(* CoDeSys 2.3 project: cy-wg-03_030.pro *)
(* Title: cy-003-wg (SanFelice) *)
(* Author: Andrea Ravasio *)
(* Libraries: serial_interface_01.lib 22.4.13 12:50:14, SerComm.lib 31.5.11 08:54:36, MBus_03.lib 22.7.15 16:25:47, Util.lib 26.9.14 10:12:46, Visual.lib 2.12.10 14:48:34, WagoLibIdent.lib 25.2.13 11:12:16, WagoLibStatus.lib 2.12.10 14:48:32, SysLibFile.lib 2.12.10 14:48:34, SysLibRtc.lib 2.12.10 14:48:32, SysLibSockets.lib 10.2.11 09:20:54, SysLibEvent.lib 2.12.10 14:48:34, SysLibPlcCtrl.lib 2.12.10 14:48:32, Standard.lib 2.12.10 14:48:34, SYSLIBCALLBACK.LIB 2.12.10 14:48:32 *)

(* PLC configuration (modules and I/O channels)
K-Bus [K_Bus] node 0, in %IB0 out %QB0
  0750-0402 4 DI 24 V DC 3.0ms [Type_1_4_Channels] node 0, in %IB24 out %QB4 {INTTypePAAssignment = PLC; INTTypeModule = plugged}
    VPN_ST2 AT %IX12.0 [BOOLOnX_I] Ch_1 Digital input
    KEY_QE_ST AT %IX12.1 [BOOLOnX_I] Ch_2 Digital input
    SCA01_5_DI AT %IX12.2 [BOOLOnX_I] Ch_3 Digital input
    PORT01_DI AT %IX12.3 [BOOLOnX_I] Ch_4 Digital input
  0750-0402 4 DI 24 V DC 3.0ms [Type_1_4_Channels] node 1, in %IB24 out %QB4 {INTTypePAAssignment = PLC; INTTypeModule = plugged}
    GAS02_DI AT %IX12.4 [BOOLOnX_I] Ch_1 Digital input
    GAS01_DI AT %IX12.5 [BOOLOnX_I] Ch_2 Digital input
    SCA01_6_DI AT %IX12.6 [BOOLOnX_I] Ch_3 Digital input
    SCA02_1_DI AT %IX12.7 [BOOLOnX_I] Ch_4 Digital input
  0750-1506 8DI / 8DO 24V DC 0.5A [Type_34_8_Channels] node 2, in %IX12.4 out %QB4 {INTTypePAAssignment = PLC; INTTypeModule = plugged}
    SCA02_2_DI AT %IX12.8 [BOOLOnX_I] Ch_1 Digital input
    SCA01_1_DO AT %QX2.0 [BOOLOnX_Q] Ch_1 Digital output
    SCA02_3_DI AT %IX12.9 [BOOLOnX_I] Ch_2 Digital input
    SCA01_2_DO AT %QX2.1 [BOOLOnX_Q] Ch_2 Digital output
    SCA02_4_DI AT %IX12.10 [BOOLOnX_I] Ch_3 Digital input
    SCA01_3_DO AT %QX2.2 [BOOLOnX_Q] Ch_3 Digital output
    SCA02_5_DI AT %IX12.11 [BOOLOnX_I] Ch_4 Digital input
    SCA01_4_DO AT %QX2.3 [BOOLOnX_Q] Ch_4 Digital output
    SCA02_6_DI AT %IX12.12 [BOOLOnX_I] Ch_5 Digital input
    AT %QX2.4 [BOOLOnX_Q] Ch_5 Digital output
    SCA02_7_DI AT %IX12.13 [BOOLOnX_I] Ch_6 Digital input
    AT %QX2.5 [BOOLOnX_Q] Ch_6 Digital output
    SCA02_8_DI AT %IX12.14 [BOOLOnX_I] Ch_7 Digital input
    AT %QX2.6 [BOOLOnX_Q] Ch_7 Digital output
    SCA02_9_DI AT %IX12.15 [BOOLOnX_I] Ch_8 Digital input
    AT %QX2.7 [BOOLOnX_Q] Ch_8 Digital output
  0750-1506 8DI / 8DO 24V DC 0.5A [Type_34_8_Channels] node 3, in %IB25 out %QB4 {INTTypePAAssignment = PLC; INTTypeModule = plugged}
    SCA03_1_DI AT %IX13.0 [BOOLOnX_I] Ch_1 Digital input
    AT %QX2.8 [BOOLOnX_Q] Ch_1 Digital output
    SCA03_2_DI AT %IX13.1 [BOOLOnX_I] Ch_2 Digital input
    AT %QX2.9 [BOOLOnX_Q] Ch_2 Digital output
    SCA03_3_DI AT %IX13.2 [BOOLOnX_I] Ch_3 Digital input
    AT %QX2.10 [BOOLOnX_Q] Ch_3 Digital output
    SCA03_4_DI AT %IX13.3 [BOOLOnX_I] Ch_4 Digital input
    AT %QX2.11 [BOOLOnX_Q] Ch_4 Digital output
    SCA03_5_DI AT %IX13.4 [BOOLOnX_I] Ch_5 Digital input
    AT %QX2.12 [BOOLOnX_Q] Ch_5 Digital output
    SCA03_6_DI AT %IX13.5 [BOOLOnX_I] Ch_6 Digital input
    AT %QX2.13 [BOOLOnX_Q] Ch_6 Digital output
    SCA03_7_DI AT %IX13.6 [BOOLOnX_I] Ch_7 Digital input
    AT %QX2.14 [BOOLOnX_Q] Ch_7 Digital output
    SCA03_8_DI AT %IX13.7 [BOOLOnX_I] Ch_8 Digital input
    AT %QX2.15 [BOOLOnX_Q] Ch_8 Digital output
  0750-1506 8DI / 8DO 24V DC 0.5A [Type_34_8_Channels] node 4, in %IB26 out %QB5 {INTTypePAAssignment = PLC; INTTypeModule = plugged}
    SCA03_9_DI AT %IX13.8 [BOOLOnX_I] Ch_1 Digital input
    AT %QX3.0 [BOOLOnX_Q] Ch_1 Digital output
    SCA03_10_DI AT %IX13.9 [BOOLOnX_I] Ch_2 Digital input
    AT %QX3.1 [BOOLOnX_Q] Ch_2 Digital output
    SCA03_11_DI AT %IX13.10 [BOOLOnX_I] Ch_3 Digital input
    AT %QX3.2 [BOOLOnX_Q] Ch_3 Digital output
    SCA03_12_DI AT %IX13.11 [BOOLOnX_I] Ch_4 Digital input
    AT %QX3.3 [BOOLOnX_Q] Ch_4 Digital output
    SCA03_13_DI AT %IX13.12 [BOOLOnX_I] Ch_5 Digital input
    AT %QX3.4 [BOOLOnX_Q] Ch_5 Digital output
    SCA03_14_DI AT %IX13.13 [BOOLOnX_I] Ch_6 Digital input
    AT %QX3.5 [BOOLOnX_Q] Ch_6 Digital output
    SCA03_15_DI AT %IX13.14 [BOOLOnX_I] Ch_7 Digital input
    AT %QX3.6 [BOOLOnX_Q] Ch_7 Digital output
    SCA03_16_DI AT %IX13.15 [BOOLOnX_I] Ch_8 Digital input
    AT %QX3.7 [BOOLOnX_Q] Ch_8 Digital output
  0750-1506 8DI / 8DO 24V DC 0.5A [Type_34_8_Channels] node 5, in %IB27 out %QB6 {INTTypePAAssignment = PLC; INTTypeModule = plugged}
    SCA03_17_DI AT %IX14.0 [BOOLOnX_I] Ch_1 Digital input
    AT %QX3.8 [BOOLOnX_Q] Ch_1 Digital output
    SCA03_18_DI AT %IX14.1 [BOOLOnX_I] Ch_2 Digital input
    AT %QX3.9 [BOOLOnX_Q] Ch_2 Digital output
    SCA03_19_DI AT %IX14.2 [BOOLOnX_I] Ch_3 Digital input
    AT %QX3.10 [BOOLOnX_Q] Ch_3 Digital output
    SCA03_20_DI AT %IX14.3 [BOOLOnX_I] Ch_4 Digital input
    AT %QX3.11 [BOOLOnX_Q] Ch_4 Digital output
    SCA03_21_DI AT %IX14.4 [BOOLOnX_I] Ch_5 Digital input
    AT %QX3.12 [BOOLOnX_Q] Ch_5 Digital output
    SCA03_22_DI AT %IX14.5 [BOOLOnX_I] Ch_6 Digital input
    AT %QX3.13 [BOOLOnX_Q] Ch_6 Digital output
    AT %IX14.6 [BOOLOnX_I] Ch_7 Digital input
    TEST1 AT %QX3.14 [BOOLOnX_Q] Ch_7 Digital output
    AT %IX14.7 [BOOLOnX_I] Ch_8 Digital input
    TEST2 AT %QX3.15 [BOOLOnX_Q] Ch_8 Digital output
  0750-0464#02 2/4 AI RTD / ADJ./ HA [Type_44_2_Channels] node 6, in %IB20 out %QB0 {INTTypePAAssignment = PLC; INTTypeModule = plugged}
    TT_S01 AT %IW0 [INTOnW_I] Ch_1 signed Input value
    AT %IW1 [INTOnW_I] Ch_2 signed Input value
  0750-0472 2 AI 0-20mA 16 Bit S.E. [Type_8_2_Channels] node 7, in %IB20 out %QB0 {INTTypePAAssignment = PLC; INTTypeModule = plugged}
    TT_S07 AT %IW2 [WORDOnW_I] I 1: Analog Input
    TT_S06 AT %IW3 [WORDOnW_I] I 2: Analog Input
  0750-0472 2 AI 0-20mA 16 Bit S.E. [Type_8_2_Channels] node 8, in %IB24 out %QB0 {INTTypePAAssignment = PLC; INTTypeModule = plugged}
    TT_S05 AT %IW4 [WORDOnW_I] I 1: Analog Input
    TT_S04 AT %IW5 [WORDOnW_I] I 2: Analog Input
  0750-0472 2 AI 0-20mA 16 Bit S.E. [Type_8_2_Channels] node 9, in %IB28 out %QB0 {INTTypePAAssignment = PLC; INTTypeModule = plugged}
    TT_S03 AT %IW6 [WORDOnW_I] I 1: Analog Input
    TT_S02 AT %IW7 [WORDOnW_I] I 2: Analog Input
  0750-0472 2 AI 0-20mA 16 Bit S.E. [Type_8_2_Channels] node 10, in %IB32 out %QB0 {INTTypePAAssignment = PLC; INTTypeModule = plugged}
    PORT01_AI AT %IW8 [WORDOnW_I] I 1: Analog Input
    AT %IW9 [WORDOnW_I] I 2: Analog Input
  0750-0650/0003-0000#03 RS 232 C Interface (Adjustable), 3 Byte [Type_21_1_Channels] node 0, in %IB36 out %QB0 {INTTypePAAssignment = PLC; INTTypeModule = plugged}
    AT %IX10.0 [BOOLOnX_I] Transmission acknowledgement
    AT %IX10.1 [BOOLOnX_I] Reception request
    AT %IX10.2 [BOOLOnX_I] Initialization acknowledgement
    AT %IX10.3 [BOOLOnX_I] Input buffer is full
    AT %IX10.4 [BOOLOnX_I] Number of received characters Bit 0
    AT %IX10.5 [BOOLOnX_I] Number of received characters Bit 1
    AT %IX10.6 [BOOLOnX_I] Number of received characters Bit 2
    AT %IB21 [BYTEOnB_I] Input data Byte 0
    AT %IB22 [BYTEOnB_I] Input data Byte 1
    AT %IB23 [BYTEOnB_I] Input data Byte 2
    AT %QX0.0 [BOOLOnX_Q] Transmission request
    AT %QX0.1 [BOOLOnX_Q] Reception acknowledgement
    AT %QX0.2 [BOOLOnX_Q] Initialization request
    AT %QX0.4 [BOOLOnX_Q] Number of characters Bit 0
    AT %QX0.5 [BOOLOnX_Q] Number of characters Bit 1
    AT %QX0.6 [BOOLOnX_Q] Number of characters Bit 2
    AT %QB1 [BYTEOnB_Q] Output data Byte 0
    AT %QB2 [BYTEOnB_Q] Output data Byte 1
    AT %QB3 [BYTEOnB_Q] Output data Byte 2
Fieldbus variables [FB_VARS] node 1, in %IB0 out %QB0
Flag variables [FLAG_VARS] node 2, in %IB0 out %QB0
Modbus-Master [MB_MASTER] node 3, in %IB0 out %QB0
*)

(* Task configuration *)
TASK FastCounter (PRIORITY := 5, INTERVAL := T#3ms);
	PLC_FAST_CTR();
END_TASK
TASK Main (PRIORITY := 10); (* freewheeling *)
	PLC_PRG();
END_TASK

(* Global variable list: Global_Constants *)
VAR_GLOBAL CONSTANT

	Plant_NAME			: STRING :='cySN:3 cyVER:30 - San Felice';
	Plant_SN			: DWORD :=3;   		(* S/N Impianto di telecontrollo *)
	Plant_SW_VER		: WORD  :=30;		(* Versione SW installata *)

	(* Parameters *)
	Plant_DefaultTAmb	: INT	:=-9999;	(* [.1°C] Temperatura ambiente di default in caso di rottura sonda *)

	(* Filesystem *)
	FilesPath  			: STRING :='S:\';

	(* TCP Logger *)
	Logger_SERVER		: STRING:='';
	Logger_IP			: STRING:='192.168.100.3';
	Logger_PORT			: WORD  :=80;
	Logger_GETSTART		: STRING:='GET /cygmsrv/hsgm.ashx?';
	Logger_GETEND		: STRING:='$R$N$R$N';
	Logger_CHECK		: STRING:='True';
	Logger_CRLF			: STRING:='$R$N';
	Logger_DataFile		: STRING:='S:\LOG.DAT';
	Logger_DataFileOld	: STRING:='S:\LOG.BCK';
	Logger_IndexFile	: STRING:='S:\LOG.IDX';
	Logger_ConnRetries	: BYTE:=5;
	Logger_RecoverMsgs	: BYTE:=100;

	(* TCP Remote *)
	Remote_PORT			: WORD  :=10;
	Remote_WELCOME		: STRING:='Connected$R$N';
	Remote_OK			: STRING:='OK$R$N';
	Remote_ERROR		: STRING:='ERROR$R$N';

	(* TCP Sockets *)
	MAX_SEND_TCP_SERVER					 : DWORD:=1500;(*60000*)
	MAX_RECEIVE_TCP_SERVER				 : DWORD:=3000;
	MAX_RECEIVE_TCP_SERVER_SOCKET	 	 : DWORD:=1500;
	MAX_SEND_TCP_CLIENT					 : DWORD:=3000;(*15000*)
	MAX_RECEIVE_TCP_CLIENT				 : DWORD:=1500;
	MAX_RECEIVE_TCP_CLIENT_SOCKET		 : DWORD:=1500;
	MAX_RECEIVE_UDP_SERVER				 : INT  :=1472;
	MAX_RECEIVE_UDP_CLIENT				 : INT  :=1472;
	CONNECT_WATCHDOG_TIME				 : TIME :=t#10s;

	(* VISU COLORS *)
	COLOR_RED 			: DWORD:=16#2020F0;
	COLOR_YELLOW		: DWORD:=16#20F0F0;
	COLOR_GREEN			: DWORD:=16#20F020;
	COLOR_GREEN_OFF 	: DWORD:=16#006000;
	COLOR_LBLUE			: DWORD:=16#F0F080;
	COLOR_GREY			: DWORD:=16#C0C0C0;

END_VAR

(* Global variable list: Global_Retain *)
VAR_GLOBAL RETAIN PERSISTENT

	PortataTotalePORT01		: DINT;
	ConteggioTotalePORT01	: DINT;
	PortataTotaleGAS01		: DINT;
	ConteggioTotaleGAS01	: DINT;
	PortataTotaleGAS02		: DINT;
	ConteggioTotaleGAS02	: DINT;

	CTB250_ENERGY_WH		: REAL;
	CTB250_ENERGY			: DWORD; (* 10^-2 MWh *)

	Mode_Manual : BOOL := FALSE;
END_VAR

(* Global variable list: Global_Variables *)
VAR_GLOBAL

	SYS    : typ_SYS;
	T_AMB  : INT;

	TPV01  : obj_TPV		:= ( ID:=1,
								 IN_EMIN:=-600 , IN_EMAX:=2500 ,
								 IN_WMIN:=-500 , IN_WMAX:=600 ); (* T_S01 *)

	TPV02  : obj_TPV_SENS	:= ( ID:=2 ,
											SogliaHL:=4096 ,   	 	(* Soglia Sonda Aperta = 2,5mA *)
											SogliaHH:=32767,	 	(* Soglia Sonda CC = 20mA *)
											SogliaWL:=10, 			(* Soglia WRN Bassa  = 10°C *)
											SogliaWH:=120,			(* Soglia WRN Alta  = 120°C *)
											PuntoMinX:=0, 		    (* Scalatura Minima vedi data di targa sonda 0°C *)
											PuntoMaxX:=160,			(* Scalatura Massima Vedi data di targa Sonda 160°C *)
											PuntoMinY:=6553,		(* Valore minimio per scalatura = 4mA *)
											PuntoMaxY:=32767,		(* Valore Massimo per Scalatura = 20mA *)
											Decimali:=1); 			(* Decimali da ottenere durante la scalatura *)
	TPV03  : obj_TPV_SENS	:= ( ID:=3 ,
											SogliaHL:=4096 ,   	 	(* Soglia Sonda Aperta = 2,5mA *)
											SogliaHH:=32767,	 	(* Soglia Sonda CC = 20mA *)
											SogliaWL:=10, 			(* Soglia WRN Bassa  = 10°C *)
											SogliaWH:=120,			(* Soglia WRN Alta  = 120°C *)
											PuntoMinX:=0, 		    (* Scalatura Minima vedi data di targa sonda 0°C *)
											PuntoMaxX:=160,			(* Scalatura Massima Vedi data di targa Sonda 160°C *)
											PuntoMinY:=6553,		(* Valore minimio per scalatura = 4mA *)
											PuntoMaxY:=32767,		(* Valore Massimo per Scalatura = 20mA *)
											Decimali:=1); 			(* Decimali da ottenere durante la scalatura *)

	TPV04  : obj_TPV_SENS	:= ( ID:=4 ,
											SogliaHL:=4096 ,   	 	(* Soglia Sonda Aperta = 2,5mA *)
											SogliaHH:=32767,	 	(* Soglia Sonda CC = 20mA *)
											SogliaWL:=10, 			(* Soglia WRN Bassa  = 10°C *)
											SogliaWH:=120,			(* Soglia WRN Alta  = 120°C *)
											PuntoMinX:=0, 		    (* Scalatura Minima vedi data di targa sonda 0°C *)
											PuntoMaxX:=160,			(* Scalatura Massima Vedi data di targa Sonda 160°C *)
											PuntoMinY:=6553,		(* Valore minimio per scalatura = 4mA *)
											PuntoMaxY:=32767,		(* Valore Massimo per Scalatura = 20mA *)
											Decimali:=1); 			(* Decimali da ottenere durante la scalatura *)

	TPV05  : obj_TPV_SENS	:= ( ID:=5 ,
											SogliaHL:=4096 ,   	 	(* Soglia Sonda Aperta = 2,5mA *)
											SogliaHH:=32767,	 	(* Soglia Sonda CC = 20mA *)
											SogliaWL:=10, 			(* Soglia WRN Bassa  = 10°C *)
											SogliaWH:=120,			(* Soglia WRN Alta  = 120°C *)
											PuntoMinX:=0, 		    (* Scalatura Minima vedi data di targa sonda 0°C *)
											PuntoMaxX:=160,			(* Scalatura Massima Vedi data di targa Sonda 160°C *)
											PuntoMinY:=6553,		(* Valore minimio per scalatura = 4mA *)
											PuntoMaxY:=32767,		(* Valore Massimo per Scalatura = 20mA *)
											Decimali:=1); 			(* Decimali da ottenere durante la scalatura *)

	TPV06  : obj_TPV_SENS	:= ( ID:=6 ,
											SogliaHL:=4096 ,   	 	(* Soglia Sonda Aperta = 2,5mA *)
											SogliaHH:=32767,	 	(* Soglia Sonda CC = 20mA *)
											SogliaWL:=10, 			(* Soglia WRN Bassa  = 10°C *)
											SogliaWH:=120,			(* Soglia WRN Alta  = 120°C *)
											PuntoMinX:=0, 		    (* Scalatura Minima vedi data di targa sonda 0°C *)
											PuntoMaxX:=160,			(* Scalatura Massima Vedi data di targa Sonda 160°C *)
											PuntoMinY:=6553,		(* Valore minimio per scalatura = 4mA *)
											PuntoMaxY:=32767,		(* Valore Massimo per Scalatura = 20mA *)
											Decimali:=1); 			(* Decimali da ottenere durante la scalatura *)

	TPV07  : obj_TPV_SENS	:= ( ID:=7 ,
											SogliaHL:=4096 ,   	 	(* Soglia Sonda Aperta = 2,5mA *)
											SogliaHH:=32767,	 	(* Soglia Sonda CC = 20mA *)
											SogliaWL:=10, 			(* Soglia WRN Bassa  = 10°C *)
											SogliaWH:=120,			(* Soglia WRN Alta  = 120°C *)
											PuntoMinX:=0, 		    (* Scalatura Minima vedi data di targa sonda 0°C *)
											PuntoMaxX:=160,			(* Scalatura Massima Vedi data di targa Sonda 160°C *)
											PuntoMinY:=6553,		(* Valore minimio per scalatura = 4mA *)
											PuntoMaxY:=32767,		(* Valore Massimo per Scalatura = 20mA *)
											Decimali:=1); 			(* Decimali da ottenere durante la scalatura *)
	(* Misuratore di Portata *)
	PORT01  : obj_PORT	:=  ( ID:=1 ,
											TempoTimeOut:=T#2m,		(* PULSE - Minuti di attesa prima di segnalare WRN di inattività sulla linea *)
											SogliaHL:=4096,   	 	(* FLOW - Soglia Sonda Aperta = 2,5mA *)
											SogliaHH:=32767,	 	(* FLOW - Soglia Sonda CC = 20mA *)
											SogliaWL:=100000, 		(* FLOW - [E-3 m3/h] Soglia WRN Bassa *)
											SogliaWH:=700000,		(* FLOW - [E-3 m3/h] Soglia WRN Alta *)
											PuntoMinX:=0, 		    (* FLOW - [E-3 m3/h] Scalatura minima vedi data di targa sonda *)
											PuntoMaxX:=800000,		(* FLOW - [E-3 m3/h] Scalatura massima Vedi data di targa sonda *)
											PuntoMinY:=6553,		(* FLOW - Valore minimio per scalatura = 4mA *)
											PuntoMaxY:=32767		(* FLOW - Valore massimo per Scalatura = 20mA *)
											);

	(*  Contatori *)
	GAS01  : obj_GAS:=  (ID:=1,	Peso:=1 ,				(* Peso del'impulso *)
								TempoTimeOut:=T#15m		(* Minuti di attesa prima di segnalare WRN di inattività sulla linea *)
													  );
	GAS02  : obj_GAS:=  (ID:=2,	Peso:=1 ,				(* Peso del'impulso *)
								TempoTimeOut:=T#15m		(* Minuti di attesa prima di segnalare WRN di inattività sulla linea *)
													  );

	(* MBUS Contabilizers *)
	MBUS01 	  : obj_MBUS				:= ( ID:=1 , COM:=2 , BAUDRATE:=BAUD_2400 );
	CTBSCAN01 : obj_MBUS_CTB_SCANNER	:= ( ID:=1 );
	(*---- MBUS DEBUG ----*)
(*	COMx					: SERIAL_INTERFACE := (bCOM_PORT_NR		:= 2,
			cbBAUDRATE			:= BAUD_2400,
			cbsBYTESIZE			:= BS_8,
			cpPARITY			:= PARITY_EVEN,
			csSTOPBITS			:= STOPBITS_1,
			cfFLOW_CONTROL		:= NO_FLOW_CONTROL);
	RXBuf					: typRING_BUFFER;
	TXBuf					: ARRAY [0..16] OF BYTE;
	xINI					: BOOL;
	xSND					: BOOL;
	maddress : BYTE;
	mchk : BYTE;
	mt1 : BOOL;
	mt2 : BOOL;
	mt3 : BOOL;
*)

	(* Virtual contabilizers *)
	CTB250	  : obj_SW_CTB				:= ( ID:=250 );

	Logger : typ_Logger;

	(**** SIMULATION ONLY ****)
	(*...*)
END_VAR

(* Data type in Errors *)
TYPE en_Logger_ErrLev :
(
	EL_Log			:=0,
	EL_Wrn			:=1,
	EL_Alarm		:=2,
	EL_AlarmStop	:=3
);
END_TYPE

(* Data type in Errors *)
TYPE en_Logger_Status :
(
	S_Logger_UNKNOWN := 0,
	S_Logger_IDLE,
	S_Logger_WAITCONN,
	S_Logger_WAITTX,
	S_Logger_WAITRESP,
	S_Logger_ERROR
);
END_TYPE

(* Data type *)
TYPE en_SYS_Objects :
(
	EO_SYS		:=0,  (* PLC *)
	EO_VPN		:=1,  (* VPN *)
	EO_DOOR		:=2,  (* Door & access control *)

	EO_CAL		:=10, (* Caldaia *)
	EO_CIR		:=11, (* Circolatore *)
	EO_CRON		:=12, (* Crono-termostato *)
	EO_VRD		:=13, (* Valvola miscelatore pannelli *)
	EO_CTL		:=14, (* Contalitri *)
	EO_CTB		:=15, (* Contabilizzatore *)
	EO_TPV		:=16, (* Temperature probes values *)
	EO_PPV		:=17, (* Pressure probes values *)
	EO_PBV		:=18, (* Over-Pressure Alarms *)
	EO_TBV		:=19, (* Over-Temperature Alarms *)
	EO_PMV		:=20, (* Under-Pressure Alarms *)
	EO_GRU		:=21, (* Gruppo termico *)
	EO_PDC		:=22, (* Pompa di calore *)
	EO_SOL		:=23, (* Pannello solare termico *)
	EO_ESOL		:=24, (* Pannello solare fotovoltaico *)
	EO_GAS		:=25, (* Contatore GAS *)
	EO_PORT		:=26, (* Misuratore di portata *)
	EO_FPV		:=27, (* Flow probes values *)
	EO_ANZ		:=28,
	EO_SCA		:=29,

	EO_LON		:=1000, (* Bus - LON *)
	EO_MODBUS	:=1001, (* Bus - MODBUS *)
	EO_MBUS		:=1002  (* Bus - M-BUS *)
);
END_TYPE

(* Data type *)
TYPE en_SYS_Status :
(
	S_UNKNOWN  := 0,
	S_STARTUP,
	S_INIT_RTC,
	S_INIT_VAR,
	S_AUTOTEST,
	S_RUNNING,
	S_SHUTDOWN,
	S_HALT
);
END_TYPE

(* Data type in Errors *)
TYPE typ_Logger :
STRUCT
	Status		: en_Logger_Status;

	SendReq		: BOOL;
	SendIdx		: DWORD;
	SendData	: ARRAY [0..MAX_SEND_TCP_CLIENT] OF BYTE;
	SendLen		: DINT;

	TData		: ARRAY [0..MAX_SEND_TCP_CLIENT] OF BYTE;
	TLen		: DINT;

	LastIdxPos	: DWORD;

	(* Temporary variables used by objects *)
	s1			: STRING(256);
	i1			: WORD;

END_STRUCT
END_TYPE

(* Data type in Plant_Objects *)
TYPE typ_MBUS_CTBS :
STRUCT
	Present			: BOOL;
	Address			: DWORD;
	NodeError		: BYTE;

	Info			: typMBusInfo;
	Data_FTemp	 	: REAL; (* C *)
	Data_RTemp	 	: REAL; (* C *)
	Data_Flow	 	: REAL; (* m3ph *)
	Data_Power	 	: REAL; (* W *)
	Data_Energy 	: REAL; (* kWh *)

	Status_Log		: BYTE;
	Status_Vis		: DWORD;

END_STRUCT
END_TYPE

(* Data type *)
TYPE typ_SYS :
STRUCT
	Status			: en_SYS_Status;
	Warning			: BOOL;
	Alarm			: BOOL;
	AlarmStop		: BOOL;

	Time_LogString	: STRING;
	Time_Year		: WORD;
	Time_Month		: BYTE;
	Time_Day		: BYTE;

	Time_CT_DT		: DT;
	Time_CT_Day		: WORD;
	Time_CT_Quarter	: BYTE;

	LastLogs_Idx	: BYTE;
	LastLogs_Dat	: ARRAY[0..5] OF STRING;
	LastLogs_Msg	: ARRAY[0..5] OF STRING;

END_STRUCT
END_TYPE

(* Data type in Plant_Objects *)
TYPE typ_VisuStrutturaMbus :
STRUCT

	sdNodoPresente: STRING(16);
	sdEnergia: STRING(16);
	sdPotenza: STRING(16);
	sdVolume: STRING(16);
	sdFlow: STRING(16);
	sdTempIngresso: STRING(8);
	sdTempaUscita: STRING(8);
	sdTempDelta: STRING(8);

END_STRUCT
END_TYPE

(* POU PLC_FAST_CTR, ST *)
PROGRAM PLC_FAST_CTR
VAR
END_VAR
GAS01.Count(Contatore:=ConteggioTotaleGAS01, Totalizzatore:=PortataTotaleGAS01);
GAS02.Count(Contatore:=ConteggioTotaleGAS02, Totalizzatore:=PortataTotaleGAS02);
END_PROGRAM

(* POU PLC_PRG, ST *)
PROGRAM PLC_PRG
VAR
	Timer1: TON; (* Fast controls tick *)
	Timer2: TON; (* Plant control tick *)
	Timer3: TON; (* Logger timer *)

	t_sum : INT; (* Vars for dynamic means of working probes *)
	t_cnt : INT;
END_VAR
(******************************************************************************
 ****                           MAIN TASK CODE                             ****
 ******************************************************************************

	Network setup:
		IP  = 192.168.100.2 | MSK = 255.255.255.0 | GW = 192.168.100.1
		DNS = 192.168.100.1 | NTP = 193.168.100.3

	Editor setup:
		Project --> Options --> Editor --> Fonts --> Courier NEW / BOLD / 12

*)

(*==============================*)
(*===== Main status machine ====*)
(*==============================*)
Main_Stm();

(*=====================================*)
(*== Running common cycle operations ==*)
(*=====================================*)
IF SYS.Status>S_INIT_VAR THEN

	(* Execute M-BUS processes *)
	MBUS01();
	CTBSCAN01( MBUS:=MBUS01 );

	GAS01 ( GAS_DI:=GAS01_DI, Totalizzatore:=PortataTotaleGAS01, Contatore:=ConteggioTotaleGAS01 );
	GAS02 ( GAS_DI:=GAS02_DI, Totalizzatore:=PortataTotaleGAS02, Contatore:=ConteggioTotaleGAS02 );

(*	COMx(	ptSEND_BUFFER		:= ADR(TXBuf),
			xSTART_SEND			:= xSND,
			utRECEIVE_BUFFER	:= RXBuf,
			xINIT				:= xINI );

	IF mt1 THEN
		mt1:=FALSE;
		COMx.iBYTES_TO_SEND:=5;
		TXBuf[0]:=16#10;
		TXBuf[1]:=16#40;
		TXBuf[2]:=maddress;
		mchk:=TXBuf[1]+TXBuf[2];
		TXBuf[3]:=mchk;
		TXBuf[4]:=16#16;
		xSND:=TRUE;
	END_IF

	IF mt2 THEN
		mt2:=FALSE;
		COMx.iBYTES_TO_SEND:=9;
		TXBuf[0]:=16#68;
		TXBuf[1]:=16#03;
		TXBuf[2]:=16#03;
		TXBuf[3]:=16#68;
		TXBuf[4]:=16#53;
		TXBuf[5]:=maddress;
		TXBuf[6]:=16#BB;
		mchk:=TXBuf[4]+TXBuf[5]+TXBuf[6];
		TXBuf[7]:=mchk;
		TXBuf[8]:=16#16;
		xSND:=TRUE;
	END_IF

	IF mt3 THEN
		mt3:=FALSE;
		COMx.iBYTES_TO_SEND:=5;
		TXBuf[0]:=16#10;
		TXBuf[1]:=16#5B;
		TXBuf[2]:=maddress;
		mchk:=TXBuf[1]+TXBuf[2];
		TXBuf[3]:=mchk;
		TXBuf[4]:=16#16;
		xSND:=TRUE;
	END_IF
*)

END_IF


(*==============================*)
(*== System cycle operations ===*)
(*==============================*)
(* Execute TCP processes *)
Logger_Proc();
Remote_Proc();
(* Update user led *)
USRLED_Update();
(* Execute Cron Editor commands *)
(*...*)
(* External resources *)
IF TPV01.ERR THEN T_AMB:=Plant_DefaultTAmb; ELSE T_AMB:=TT_S01; END_IF

(**** SIMULATION ONLY ****)
(*...*)
END_PROGRAM
ACTION Main_Stm:
CASE Sys.Status OF
	(*--------------------------------------------------------*)
	S_STARTUP:
		Sys.Status:=S_INIT_RTC;
	(*--------------------------------------------------------*)
	S_INIT_RTC:
		(* Check RTC and update from network *)
		RTC_Update();
		(* Check time *)
		IF Sys.Time_Year>2000 THEN
			Sys.Status:=S_INIT_VAR;
		END_IF
	(*--------------------------------------------------------*)
	S_INIT_VAR:
		LogEv(EL_Wrn,EO_SYS,0,1,CONCAT('System_startup_v',WORD_TO_STRING(Plant_SW_VER)));
		Sys.Status:=S_RUNNING;
	(*--------------------------------------------------------*)
	S_RUNNING:

		Timer1(IN:=NOT Timer1.Q,PT:=T#150ms);
		IF Timer1.Q THEN
			(* Update system checks *)
			SCA_Proc();
			SYS_Proc();
		END_IF

		Timer2(IN:=NOT Timer2.Q,PT:=T#500ms);
		IF Timer2.Q THEN
			(* Read current date/time *)
			RTC_Update();
			(* === Execute plant operations === *)
			(* Temperature da RTD *)
			TPV01	 ( IN:=TT_S01 );
			(* Temperature da Convertitori 4-20mA *)
			TPV02	 ( AI_INPUT:=TT_S02 );
			TPV03	 ( AI_INPUT:=TT_S03 );
			TPV04	 ( AI_INPUT:=TT_S04 );
			TPV05	 ( AI_INPUT:=TT_S05 );
			TPV06	 ( AI_INPUT:=TT_S06 );
			TPV07	 ( AI_INPUT:=TT_S07 );
			(* Contabilizzatori Digitali *)
				(* Media dinamica delle temperature valide *)
				t_sum:=0; t_cnt:=0;
				IF NOT TPV02.ERR THEN t_sum:=t_sum+TPV02.ValoreScalato; t_cnt:=t_cnt+1; END_IF
				IF NOT TPV03.ERR THEN t_sum:=t_sum+TPV03.ValoreScalato; t_cnt:=t_cnt+1; END_IF
				IF NOT TPV04.ERR THEN t_sum:=t_sum+TPV04.ValoreScalato; t_cnt:=t_cnt+1; END_IF
				IF t_cnt>0 THEN CTB250.T_SEND:=t_sum/t_cnt; ELSE CTB250.T_SEND:=-9999; END_IF
				t_sum:=0; t_cnt:=0;
				IF NOT TPV05.ERR THEN t_sum:=t_sum+TPV05.ValoreScalato; t_cnt:=t_cnt+1; END_IF
				IF NOT TPV06.ERR THEN t_sum:=t_sum+TPV06.ValoreScalato; t_cnt:=t_cnt+1; END_IF
				IF NOT TPV07.ERR THEN t_sum:=t_sum+TPV07.ValoreScalato; t_cnt:=t_cnt+1; END_IF
				IF t_cnt>0 THEN CTB250.T_RET:=t_sum/t_cnt; ELSE CTB250.T_RET:=-9999; END_IF
				(* Ferma contabilizzazione se manca una temperatura *)
				IF CTB250.T_SEND=-9999 OR CTB250.T_RET=-9999 THEN CTB250.T_SEND:=0; CTB250.T_RET:=0; END_IF
			CTB250   (	FLOW  :=PORT01.ValoreScalato,
						ENERGY_WH:=CTB250_ENERGY_WH,
						ENERGY   :=CTB250_ENERGY );

			(* Test toggle *)
			IF TEST1 THEN TEST1:=FALSE; ELSE TEST1:=TRUE; END_IF
		     END_IF

		Timer3(IN:=NOT Timer3.Q,PT:=T#5m);
		IF Timer3.Q THEN
			(* Trig logger *)
			LogTrig();
			(* Execute temporary CSV logger *)
			CSV_Log();
		END_IF

		(* Contabilizzatori Digitali *)
		PORT01( DI_Input:=PORT01_DI, AI_INPUT:=PORT01_AI,
				Totalizzatore:=PortataTotalePORT01,
				Contatore:=ConteggioTotalePORT01 );


	(*--------------------------------------------------------*)
	S_SHUTDOWN:
		(* Arresto del sistema *)
		Sys.Status:=S_STARTUP;
	(*--------------------------------------------------------*)
	S_HALT:
		(* Aspetta uscita manuale *)
		Sys.Status:=S_STARTUP;
	(*--------------------------------------------------------*)
ELSE
	Sys.Status:=S_STARTUP;
END_CASE;
END_ACTION

(* POU TCP_Logger/Logger_Proc, ST *)
PROGRAM Logger_Proc
VAR
	c1:         	TCPCLIENT;

	Open:	    	BOOL;
	IpAddr:			DWORD;
	InetAddr:		DWORD;
	Connected:  	BOOL;
	Error:      	DINT;
	TxTrig:     	BOOL;
	RxData:			ARRAY [0..MAX_RECEIVE_TCP_CLIENT] OF BYTE;
	RxLen:			DINT;

	Retry:			BYTE;	(* Counter for connection retries *)
	Recovered:		BYTE;	(* Counter for recovered unsent messages *)

	i:				DINT;
	pos:			DWORD;
	hFile:			DWORD;

END_VAR
(*=== State machine ===*)
CASE Logger.Status OF

	S_Logger_UNKNOWN:
		(* Startup *)
		Logger.SendReq:=FALSE;
		Open:=FALSE;
		Logger.Status:=S_Logger_IDLE;

	S_Logger_IDLE:
		(* Wait request *)
		IF Logger.SendReq THEN
			(* Resolve server name or use static IP *)
			IF LEN(Logger_SERVER)=0 THEN
				InetAddr:=SysSockInetAddr(Logger_IP);
			ELSE
				IpAddr:=SysSockGetHostByName(ADR(Logger_SERVER));
				DWORDSWAP(pIn:=ADR(IpAddr), pOut:=ADR(InetAddr));
			END_IF
			TxTrig:=FALSE;
			RxLen:=0;
			(* Open connection *)
			Open:=TRUE;
			Logger.Status:=S_Logger_WAITCONN;
		END_IF

	S_Logger_WAITCONN:
		(* Wait connection *)
		IF Connected THEN
			(* Send data *)
			TxTrig:=TRUE;
			Logger.Status:=S_Logger_WAITTX;
		END_IF
		IF Error>0 THEN
			Open:=FALSE;
			Logger.Status:=S_Logger_ERROR;
		END_IF

	S_Logger_WAITTX:
		(* Wait transmission *)
		IF NOT TxTrig THEN
			Logger.Status:=S_Logger_WAITRESP;
		END_IF
		IF Error>0 THEN
			Open:=FALSE;
			Logger.Status:=S_Logger_ERROR;
		END_IF

	S_Logger_WAITRESP:
		(* Wait response *)
		IF Connected=FALSE (* OR TIMEOUT!! *) THEN
			Open:=FALSE;
			(* Check response *)
			IF RxLen>=4 AND CHKSTRING(pString:=ADR(RxData), pPattern:=ADR(Logger_CHECK)) THEN
				Logger.SendReq:=FALSE;
				Retry:=0;
				(* Check unsent messages to flush *)
				IF Recovered<Logger_RecoverMsgs THEN
					MsgChk();
					IF Logger.SendReq=TRUE THEN
						Recovered:=Recovered+1;
					ELSE
						Recovered:=0;
					END_IF
				ELSE
					Recovered:=0;
				END_IF
				Logger.Status:=S_Logger_IDLE;
			ELSE
				Logger.Status:=S_Logger_ERROR;
			END_IF
		END_IF

	S_Logger_ERROR:
		(* Connection error or send failure *)
		Retry:=Retry+1;
		IF Retry>Logger_ConnRetries THEN
			(* Save message as unsent *)
			MsgSave();
			Logger.SendReq:=FALSE;
			Retry:=0;
		END_IF
		Logger.Status:=S_Logger_IDLE;

ELSE
	Logger.Status:=S_Logger_UNKNOWN;
END_CASE


(*=== Execute client lib ===*)
c1(
	xOpenConnection			:= Open,
	dwInetAddr 				:= InetAddr,
	wPortNumber				:= Logger_PORT,
	ptSendData				:= ADR(Logger.SendData),
	diSendCount				:= Logger.SendLen,
	tConnectWatchdogTime	:= t#10s,
	xStartSend				:= TxTrig,
	aReceiveBuffer			:= RxData,
	diReceiveCount			:= RxLen,
	xConnected				=> Connected,
	diError					=> Error
);

(*=== Process Rx data ===*)
(*IF RxLen>0 THEN
	RxLen:=0;
END_IF*)
END_PROGRAM
ACTION MsgChk:
(* Open index file *)
hFile:=SysFileOpen(Logger_IndexFile,'r');
IF hFile=0 THEN
	RETURN;
END_IF
(* Search oldest message to recover *)
SysFileSetPos(hFile,Logger.LastIdxPos);
Logger.SendLen:=0;
REPEAT
	SysFileRead(hFile, ADR(Logger.SendIdx), SIZEOF(Logger.SendIdx));
	pos:=SysFileGetPos(hFile);
	SysFileRead(hFile, ADR(Logger.SendLen), SIZEOF(Logger.SendLen));
UNTIL
	SysFileEOF(hFile) OR Logger.SendLen<>0
END_REPEAT
SysFileClose(hFile);
(* Delete index file when all messages are recovered *)
IF Logger.SendLen=0 THEN
	Logger.LastIdxPos:=0;
	SysFileDelete(Logger_IndexFile);
	RETURN;
END_IF
(* Recover message data *)
hFile:=SysFileOpen(Logger_DataFile,'r');
IF hFile<>0 THEN
	SysFileSetPos(hFile,Logger.SendIdx);
	SysFileRead(hFile,ADR(Logger.SendData),Logger.SendLen);
	Logger.SendReq:=TRUE;
	SysFileClose(hFile);
END_IF
(* Clear index entry *)
hFile:=SysFileOpen(Logger_IndexFile,'a');
IF hFile<>0 THEN
	SysFileSetPos(hFile,pos);
	i:=0;
	SysFileWrite(hFile, ADR(i), 4);
	Logger.LastIdxPos:=SysFileGetPos(hFile);
	SysFileClose(hFile);
END_IF
END_ACTION
ACTION MsgSave:
(* Add log position in recovery indexes *)
hFile:=SysFileOpen(Logger_IndexFile,'a');
SysFileWrite(hFile, ADR(Logger.SendIdx), SIZEOF(Logger.SendIdx));
SysFileWrite(hFile, ADR(Logger.SendLen), SIZEOF(Logger.SendLen));
SysFileClose(hFile);
END_ACTION

(* POU Utils Functions/TCPCLIENT, ST *)
FUNCTION_BLOCK TCPCLIENT
(***********************************************************************************************************	*)
(* Version: 1.3b                        			          													*)
(* Date: 28.10.2014                   				          							            			*)
(***********************************************************************************************************	*)
(* WAGO Kontakttechnik GmbH Hansastr. 27 32423 Minden(Westf.)													*)
(* Tel. +0049 571/887-0 Fax. +0049 571/887-0																	*)
(* Author: VB																									*)
(***********************************************************************************************************	*)
(*Description:	A TCP client to read and write data with additional connection watchdog							*)
(*History:																										*)
(*Version 1.3b: 28.10.2014: Use DWORD address for IP (Andrea Ravasio)											*)
(*Version 1.3: 11.02.2011: Changes according to 750-880/881											 			*)
(*Version 1.2: 29.08.2007 Bugfix TCP Client																		*)
(*Version 1.1: 15.01.2007 Changes according to FW11																*)
(*Version 1.0: 09.03.2006 Release																				*)
(***********************************************************************************************************	*)
VAR CONSTANT
	STATE_CREATE     				 : BYTE:= 0;
	STATE_OPEN     					 : BYTE:= 1;
	STATE_IOCTL    					 : BYTE:= 2;
	STATE_CONNECT     				 : BYTE:= 10;
	STATE_TX       					 : BYTE:= 20;
	STATE_RX       					 : BYTE:= 30;
	STATE_CLOSE    					 : BYTE:= 40;
	STATE_ERROR_TRAP			     : BYTE:= 200;
END_VAR

VAR_INPUT
	xOpenConnection					: BOOL;
	dwInetAddr						: DWORD; (* <== Use SysSockInetAddr() value or
													swapped bytes order of SysSockGetHostByName() value *)
	wPortNumber						: WORD;
	ptSendData						: POINTER TO ARRAY[0..MAX_SEND_TCP_CLIENT] OF BYTE;
	diSendCount						: DINT;
	tConnectWatchdogTime		    : TIME := t#10s;
END_VAR
VAR_OUTPUT
	xConnected						: BOOL;
	diError 						: DINT := 0;
END_VAR
(* ErrorCodes -----------------------------------------
	16#8001 => No socket descriptor available 
	16#8002 => SysSockSend returns -1 
	16#8003 => Socket was "gracefully closed" 
	16#8004 => switching to none blocking mode fails
	16#8005 => SysSockClose() returns FALSE 
    16#8006 => SysSockConnect() fails
    16#8007 => SysSockSend() fails
	16#8008 => error state machine 
	16#8009 => timeout while waiting for data from server 
------------------------------------------------------------*)
VAR_IN_OUT
	xStartSend							: BOOL;
	aReceiveBuffer						: ARRAY [0..MAX_RECEIVE_TCP_CLIENT] OF BYTE;
	diReceiveCount						: DINT;
END_VAR
VAR
	m_State								: BYTE := 0;
	m_ReceiveBuffer						: ARRAY [0..MAX_RECEIVE_TCP_CLIENT_SOCKET] OF BYTE;
	m_Socket							: DINT;
	m_AddressInfo						: SOCKADDRESS;
	m_BytesReceived						: DINT;
	m_diReturn							: DINT;
	m_xReturn							: BOOL;
	m_IoCtlParameter  					: DINT := 1; (* IOCTL-Parameter for non-blocking mode of sockets *)
	i									: INT;
	T_Connect							: TON;
	m_count								: DINT;
	diOption							: DINT := 1;
	m_Blocking   						: DINT := 0;
END_VAR
IF xOpenConnection THEN
	(* State maschine *)
	CASE  m_State OF

	(* -------------------------------------------------------------------------*)
	STATE_CREATE:
			(* create socket descriptor*)
			m_Socket := SysSockCreate(diAddressFamily	:= SOCKET_AF_INET,
													 diType		:= SOCKET_STREAM,
													 diProtocol := SOCKET_IPPROTO_TCP);
			IF m_Socket >= 0 THEN
			(*Set Push-Bit*)
				IF ADR(%MW0)=16#30000000  OR ADR(%MW0)=16#20000000 THEN (*841 or 881*)
					SysSockSetOption(
						diSocket:=m_Socket,
						diLevel:=6,
						diOption:=SOCKET_TCP_NODELAY,
						pOptionValue:=ADR(diOption),
						diOptionLength:=SIZEOF(diOption));
				ELSE
						;
				END_IF
				m_State := STATE_IOCTL; (* succesful *)
			ELSE
				diError := 16#8001;  (* no socket descriptor available *)
				m_State := STATE_ERROR_TRAP;
			END_IF

	(* -------------------------------------------------------------------------*)
	STATE_IOCTL: (* change  socket mode  to none blocking *)
		m_diReturn := SysSockIoctl( m_Socket, SOCKET_FIONBIO, ADR(m_IoCtlParameter));
		IF m_diReturn <> 0 THEN
			m_AddressInfo.sin_family := SOCKET_AF_INET;
			m_AddressInfo.sin_port := SysSockNtohs(wPortNumber);
			m_AddressInfo.sin_addr := dwInetAddr;
			m_State := STATE_CONNECT;
		ELSE
			diError := 16#8004;  (* switching to none blocking mode fails *)
			m_State := STATE_ERROR_TRAP;
		END_IF


	(* -------------------------------------------------------------------------*)
	STATE_CONNECT: (* connect with server *)
		T_Connect(IN:=TRUE , PT:=tConnectWatchdogTime);(*activate watchdog for establishing connection to a server*)
		m_xReturn := SysSockConnect ( m_Socket, ADR(m_AddressInfo),  SIZEOF(m_AddressInfo));
		IF m_xReturn THEN (* succesful *)
			IF xStartSend THEN
				m_State := STATE_TX;(*transmit data*)
			ELSE
				m_State := STATE_RX;(*wait for data from server*)
			END_IF
			xConnected:=TRUE;
			T_Connect(IN:=FALSE);
		ELSE
			IF T_Connect.Q THEN
				diError := 16#8006;  (* connect fails *)
				xConnected:=FALSE;
				T_Connect(IN:=FALSE);
				m_State := STATE_ERROR_TRAP;
				SysSockClose( m_Socket);
			ELSE
				m_State := STATE_CONNECT;(*client still  tries to set up connection*)
			END_IF
		END_IF


	STATE_TX:	 (* send TCP-message *)
		m_diReturn := SysSockSend(diSocket := m_Socket,
								  pbyBuffer := ADR(ptSendData^[0]),
								  diBufferSize := diSendCount-m_count,
								  diFlags := 0);

		CASE m_diReturn OF
		-1:	(* ERROR *)
			T_Connect(IN:=TRUE , PT:=CONNECT_WATCHDOG_TIME);(*activate watchdog to check communication*)
			IF t_Connect.Q THEN
				diError := 16#8007;
				T_Connect(IN:=FALSE);
				m_State:=STATE_CLOSE;
			END_IF
		0: (* socket was "gracefully closed" *)
			m_State := STATE_CLOSE;
			diError := 16#8003;
		ELSE (* succesful *)
			m_count:=m_count+m_diReturn;
			IF m_count>=diSendCount THEN
				diError := 16#0000;
				m_State := STATE_RX;
				m_count:=0;
				xStartSend:=FALSE;
			END_IF
			T_Connect(IN:=FALSE);
		END_CASE

	(* -------------------------------------------------------------------------*)
	STATE_RX: (* process receive data *)
			m_BytesReceived := SysSockRecv(	diSocket 	:= m_Socket,
										pbyBuffer 	:= ADR(m_ReceiveBuffer),		(* Address of receive buffer *)
										diBufferSize:= SIZEOF(m_ReceiveBuffer),
										diFlags		:= 0);

			CASE m_BytesReceived OF
			-1:	(* No data available or error occured *)
				T_Connect(IN:=TRUE , PT:=tConnectWatchdogTime);(*activate watchdog to check communication*)
				IF t_Connect.Q THEN
					diError:=16#8009;
					T_Connect(IN:=FALSE);
					m_State:=STATE_CLOSE;
				END_IF
				IF xStartSend THEN
					m_State:=STATE_TX	;(* WAIT IN THIS STATE  and check for arriving data or new send command*)
				END_IF;
			0: (* socket was "gracefully closed"  *)
				m_State:=STATE_CLOSE;
				diError := 16#8003;
			ELSE (* succesful *)
				diError := 16#0000;
				T_Connect(IN:=FALSE);
				(* Copy received data into receive buffer *)
				FOR i:= 0 TO DINT_TO_INT(m_BytesReceived	)-1 DO
					aReceiveBuffer[diReceiveCount]:= m_ReceiveBuffer[i];
					diReceiveCount:=(diReceiveCount+1) MOD SIZEOF(aReceiveBuffer);
				END_FOR

			END_CASE

	(* -------------------------------------------------------------------------*)
	STATE_CLOSE : (* close socket *)
		IF ADR(%MW0)=16#30000000  OR ADR(%MW0)=16#20000000 THEN (*841 or 881*)
			;
		ELSE
			SysSockShutdown(m_Socket, 0);;(*870*)
		END_IF
		m_xReturn := SysSockClose( m_Socket);
		m_Socket := -1;
		m_State := 0; (* succesful *)
		xConnected:=FALSE;
		T_Connect(IN:=FALSE);
	(* -------------------------------------------------------------------------*)
	STATE_ERROR_TRAP: (* error handling *)
		xConnected:=FALSE;

	ELSE  (* Bad FSM code trap  *)
			m_State:= STATE_ERROR_TRAP;
			diError:= 16#8008;
	END_CASE

ELSE(*close connection*)
	IF m_Socket >= 0 THEN
		IF ADR(%MW0)=16#30000000  OR ADR(%MW0)=16#20000000 THEN (*841 or 881*)
			;
		ELSE
			SysSockShutdown(m_Socket, 0);;(*870*)
		END_IF
		SysSockClose( m_Socket);
	END_IF
	m_Socket := -1;
	diError := 16#0000;
	m_State := STATE_CREATE;
	xConnected:=FALSE;
	T_Connect(IN:=FALSE);
END_IF
END_FUNCTION_BLOCK

(* POU Utils Functions/DWORDSWAP, ST *)
FUNCTION DWORDSWAP:BOOL
VAR_INPUT
	pIn:POINTER TO ARRAY[1..4] OF BYTE;
	pOut:POINTER TO ARRAY[1..4] OF BYTE;
END_VAR
VAR
END_VAR
pOut^[1]:=pIn^[4];
pOut^[2]:=pIn^[3];
pOut^[3]:=pIn^[2];
pOut^[4]:=pIn^[1];
END_FUNCTION

(* POU Utils Functions/CHKSTRING, ST *)
FUNCTION CHKSTRING : BOOL
VAR_INPUT
	pString: POINTER TO BYTE;
	pPattern: POINTER TO BYTE;
END_VAR
VAR
END_VAR
CHKSTRING:=TRUE;
WHILE pPattern^<>0 AND CHKSTRING DO
	IF pPattern^<>pString^ THEN CHKSTRING:=FALSE; END_IF
	pString:=pString+1;
	pPattern:=pPattern+1;
END_WHILE
END_FUNCTION

(* POU TCP_Remote/Remote_Proc, ST *)
PROGRAM Remote_Proc
VAR
	s1:         	TCPSERVER;
	Enable: 		BOOL;
	Connected: 		BOOL;
	Error: 			DINT;

	TxData:			ARRAY [0..MAX_SEND_TCP_SERVER] OF BYTE;
	TxLen:			DINT;
	TxTrig:			BOOL;

	RxData:			ARRAY [0..MAX_RECEIVE_TCP_SERVER] OF BYTE;
	RxLen:			DINT;

	Status:			DINT;

	(* Command interpreter *)

	Cmd_Buf:		ARRAY [0..MAX_RECEIVE_TCP_SERVER] OF BYTE;
	Cmd_Buf_U16:	POINTER TO WORD;
	Cmd_Buf_INT:	POINTER TO INT;
	Cmd_BufLen:		WORD;
	Cmd_St:			WORD;

	Cmd_Obj:		WORD;
	Cmd_ObjIdx:		WORD;
	Cmd_C:			WORD;
	Cmd_R:			WORD;
	Cmd_CLen:		WORD;
	Cmd_RLen:		WORD;

	i : WORD;
	j : INT;

END_VAR
(*=== State machine ===*)
CASE Status OF
	0: (* Startup *)
		TxLen:=0; TxTrig:=FALSE;
		RxLen:=0;
		Enable:=TRUE;
		Status:=1;

	1: (* Wait incoming connection *)
		IF Connected THEN
			(* Log access *)
			LogEv(EL_Log,EO_VPN,1,5,'Remote');
			(* Send welcome message *)
			(*ADDSTRING(pTxData:=ADR(TxData), pString:=ADR(Remote_WELCOME), TxLen:=TxLen);
			TxTrig:=TRUE;*)
			Cmd_BufLen:=0;
			Cmd_St:=0;
			Status:=2;
		END_IF
		IF Error>1 THEN
			Enable:=FALSE;
			Status:=0;
		END_IF

	2: (* Wait command *)
		IF RxLen>0 THEN
			(*=== Interpreter start ===*)
			IF Cmd_BufLen+(RxLen/2)>=MAX_RECEIVE_TCP_SERVER THEN
				(* ERROR *)
				Cmd_BufLen:=0;
			ELSE
				i:=HEXTORAW(pString:=ADR(RxData), StringLen:=DINT_TO_WORD(RxLen), pData:=ADR(Cmd_Buf[Cmd_BufLen]));
				Cmd_BufLen:=Cmd_BufLen+i;
			END_IF
			IF Cmd_BufLen>=8 THEN
				Cmd_Buf_U16:=ADR(Cmd_Buf[6]);
				IF Cmd_BufLen>=(8+Cmd_Buf_U16^) THEN
					Cmd_CLen:=Cmd_Buf_U16^;
					Cmd_Buf_U16:=ADR(Cmd_Buf[0]); Cmd_Obj:=Cmd_Buf_U16^;
					Cmd_Buf_U16:=ADR(Cmd_Buf[2]); Cmd_ObjIdx:=Cmd_Buf_U16^;
					Cmd_Buf_U16:=ADR(Cmd_Buf[4]); Cmd_C:=Cmd_Buf_U16^;
					Command();
					Cmd_BufLen:=0;
				END_IF
			END_IF
			(*=== Interpreter end ===*)
			RxLen:=0;
		END_IF
		IF NOT Connected THEN
			Status:=0;
		END_IF

ELSE
	Status:=0;
END_CASE


(*=== Execute server lib ===*)
s1(
	xEnable				:= Enable,
	wPortNumber			:= Remote_PORT,
	tServerTimeOut		:= t#15m,
	ptSendData			:= ADR(TxData),
	diSendCount			:= TxLen,
	xStartSend			:= TxTrig,
	aReceiveBuffer		:= RxData,
	diReceiveCount		:= RxLen,
	xClientConnected	=> Connected,
	diError				=> Error
);
END_PROGRAM
ACTION Cmd_CTB:
(* Check index *)
IF Cmd_ObjIdx<>1 THEN
	Cmd_R:=2;
	RETURN;
END_IF

(* Process command *)
CASE Cmd_C OF

	1: (* START REFRESH *)
		CTBSCAN01.Refresh:=TRUE;
	2: (* START REFRESH *)
		CTBSCAN01.Refresh:=FALSE;
	3: (* START RESCAN/SEARCH *)
		CTBSCAN01.Rescan:=TRUE;
	4: (* STOP  RESCAN/SEARCH *)
		CTBSCAN01.Rescan:=FALSE;

ELSE
	Cmd_R:=3;
END_CASE
END_ACTION
ACTION Cmd_SYS:
(* Check index *)
IF Cmd_ObjIdx<>0 THEN
	Cmd_R:=2;
	RETURN;
END_IF

(* Process command *)
CASE Cmd_C OF

	0: (* ECHO *)
		IF Cmd_CLen<>0 THEN
			TxLen:=0;
		END_IF

	1: (* LOG REQUEST *)
		LogTrig();

	2: (* REARM *)
		Sys.Warning:=FALSE;
		Sys.Alarm:=FALSE;
		Sys.AlarmStop:=FALSE;

ELSE
	Cmd_R:=3;
END_CASE
END_ACTION
ACTION Command:
(* Default response OK/NODATA *)
Cmd_R:=0;
Cmd_RLen:=0;
TxLen:=16;

(* Check object *)
CASE Cmd_Obj OF

	EO_SYS:
		Cmd_SYS();

	EO_CTB:
		Cmd_CTB();

ELSE
	Cmd_R:=1;
END_CASE

(* Generate response *)
IF TxLen>0 THEN
	RAWTOHEX(ADR(Cmd_Obj)	,2,ADR(TxData[ 0]));
	RAWTOHEX(ADR(Cmd_ObjIdx),2,ADR(TxData[ 4]));
	RAWTOHEX(ADR(Cmd_R)		,2,ADR(TxData[ 8]));
	RAWTOHEX(ADR(Cmd_RLen)	,2,ADR(TxData[12]));
	TxTrig:=TRUE;
END_IF
END_ACTION

(* POU Utils Functions/TCPSERVER, ST *)
FUNCTION_BLOCK TCPSERVER
(***********************************************************************************************************	*)
(* Version: 1.6                                    			          											*)
(* Date: 11.02.2011                                   					          							    *)
(***********************************************************************************************************	*)
(* WAGO Kontakttechnik GmbH Hansastr. 27 32423 Minden(Westf.)													*)
(* Tel. +0049 571/887-0 Fax. +0049 571/887-0																	*)
(* Author: VB																									*)
(***********************************************************************************************************	*)
(*Description:	A TCP server to read and write data													       		*)
(*Historie:																										*)
(*Version 1.6: 11.02.2011: Changes according to 750-880/881											 			*)
(*Version 1.5: 27.11.2008 Bugfix allow reuse port																*)
(*Version 1.4: 13.10.2008 Bugfix transmitting large data														*)
(*Version 1.3: 15.01.2007 Changes according to FW11																*)
(*Version 1.2: 09.03.2006 Changes for socket handle 0											       			*)
(*Version 1.1: 14.02.2005 Release																				*)
(***********************************************************************************************************	*)
VAR CONSTANT
	STATE_INIT     				 : BYTE:= 0;
	STATE_OPEN     				 : BYTE:= 1;
	STATE_TX       				 : BYTE:= 20;
	STATE_RX       				 : BYTE:= 30;
	STATE_CLOSE    				 : BYTE:= 40;
	STATE_ERROR_TRAP		 	 : BYTE:= 200;
END_VAR
VAR_INPUT
	xEnable    					: BOOL;	 (* Set TRUE to enable function block *)
	wPortNumber					: WORD;  (* Port *)
	tServerTimeOut				: TIME:=t#50s;
	ptSendData					: POINTER TO ARRAY[0..MAX_SEND_TCP_SERVER] OF BYTE;
	diSendCount					: DINT;
END_VAR
VAR_OUTPUT
	xClientConnected  			: BOOL:= FALSE;
	diError 					: DINT:= 0;
END_VAR
(* Status Codes -----------------------------------------
	16#8001 => No socket descriptor available 
	16#8002 => SysSockBind fails 
	16#8003 => SysSockListen fails 
	16#8004 => switching to none blocking mode fails
	16#8005 => SysSockClose() returns FALSE 
    16#8006 => SysSockConnect() fails
    16#8007 => SysSockSend() fails
	16#8008 => error state machine 
	16#8009 => timeout while waiting for data from server 
	16#0001 => server waiting for client to establish connection
------------------------------------------------------------*)
VAR_IN_OUT
	xStartSend					: BOOL;
	aReceiveBuffer				: ARRAY [0..MAX_RECEIVE_TCP_SERVER] OF BYTE;
	diReceiveCount				: DINT;
END_VAR

VAR
	m_State    					: BYTE:= 0;
	m_ReceiveBuffer				: ARRAY [0..MAX_RECEIVE_TCP_SERVER_SOCKET] OF BYTE;
	m_ServerSocket				: DINT:= SOCKET_INVALID;
	m_Socket					: DINT:= SOCKET_INVALID;
	m_AddressInfo				: SOCKADDRESS;
	m_BytesReceived				: DINT;
	m_diReturn					: DINT;
	m_xReturn					: BOOL;
	m_SizeSockadr				: DWORD;
	m_ConnectionWatchdog		: TON;
	m_Flags						: DINT;
	m_NoneBlocking   			: DINT:= 1;
	m_Blocking   				: DINT:= 0;
	i							: INT;
	m_count						: DINT;
	diOption					: DINT := 1;
	on: DINT;
END_VAR
IF xEnable THEN
	CASE m_State OF
		STATE_INIT:
			(* Create Socket *)
			m_ServerSocket:= SysSockCreate( SOCKET_AF_INET, SOCKET_STREAM, 0);
			IF m_ServerSocket = SOCKET_INVALID THEN
				(* *)
				diError:= 16#8001;
				m_State:= STATE_ERROR_TRAP;
				RETURN;
			ELSE
				;
			END_IF
			(* Address bindings *)
			(********************)
			on:=1;
			SysSockSetOption( m_ServerSocket, SOCKET_SOL, SOCKET_SO_REUSEADDR, ADR(on), SIZEOF(on) );

			m_AddressInfo.sin_family:= SOCKET_AF_INET;
			m_AddressInfo.sin_port  := SysSockHtons( wPortNumber);
			m_AddressInfo.sin_addr  := SOCKET_INADDR_ANY;
			IF NOT SysSockBind( m_ServerSocket, ADR(m_AddressInfo), SIZEOF(m_AddressInfo)) THEN
				diError:= 16#8002;
				m_State:= STATE_ERROR_TRAP;
				RETURN;
			END_IF
			(* Wait for connections *)
			(************************)
			IF NOT SysSockListen( m_ServerSocket, 1) THEN
				diError:= 16#8003;
				m_State:= STATE_ERROR_TRAP;
			END_IF

			(* Puts SOCKET in NonBlocking mode *)
			m_diReturn:= SysSockIoctl( m_ServerSocket, SOCKET_FIONBIO, ADR(m_NoneBlocking));

			m_State:= STATE_OPEN;


		STATE_OPEN: 	(* Waiting for incomming connection *)
				m_SizeSockadr:=SIZEOF(m_AddressInfo);
				m_Socket:= SysSockAccept( m_ServerSocket, ADR(m_AddressInfo), ADR(m_SizeSockadr));
				diError:=State_open;
				IF m_Socket <> SOCKET_INVALID THEN
					xClientConnected:=TRUE;
					(*Set Push-Bit:new V1.5*)
					IF ADR(%MW0)=16#30000000  OR ADR(%MW0)=16#20000000 THEN (*841 or 881*)
						SysSockSetOption(
							diSocket:=m_Socket,
							diLevel:=6,
							diOption:=SOCKET_TCP_NODELAY,
							pOptionValue:=ADR(diOption),
							diOptionLength:=SIZEOF(diOption));
					ELSE
							;
					END_IF
					SysSockIoctl( m_Socket, SOCKET_FIONBIO, ADR(m_NoneBlocking));
					m_State:= STATE_RX;
					diError:=0;
				END_IF

		STATE_RX:
					m_BytesReceived:= SysSockRecv( m_Socket, ADR(m_ReceiveBuffer), SIZEOF(m_ReceiveBuffer), 0);
					CASE m_BytesReceived OF
					-1:(*no data available or error occured*)
						m_ConnectionWatchdog(IN:=TRUE , PT:=tServerTimeOut );
						IF m_connectionWatchdog.Q THEN
							m_State:= STATE_CLOSE;
							m_ConnectionWatchdog(IN:=FALSE);(*reset connection watchdog*)
							diError := 16#8009;
						END_IF
					0:(* socket was "gracefully closed"  *)
						m_State:= STATE_CLOSE;
						diError := 16#8003;
					ELSE
						(* Copy received data into receive buffer *)
						(********************************)
						FOR i:= 0 TO DINT_TO_INT(m_BytesReceived	)-1 DO
							aReceiveBuffer[diReceiveCount]:= m_ReceiveBuffer[i];
							diReceiveCount:=(diReceiveCount+1) MOD SIZEOF(aReceiveBuffer);
						END_FOR

						m_ConnectionWatchdog(IN:=FALSE);(*reset connection watchdog*)
					END_CASE

				(*send data*)
				IF xStartSend	 THEN
					m_State := STATE_TX;
				END_IF

	STATE_TX:	 (* send TCP-message *)
		m_diReturn := SysSockSend(diSocket := m_Socket,
								  pbyBuffer := ADR(ptSendData^[m_count]),(*geändert V1.4 bisher: [0] *)
								  diBufferSize := diSendCount-m_count,
								  diFlags :=m_Flags);
		CASE m_diReturn OF
		-1:	(* ERROR or data could not yet be send (V1.3 due to new FW11) *)
			m_ConnectionWatchdog(IN:=TRUE , PT:=tServerTimeOut );
			IF m_connectionWatchdog.Q THEN
				m_State:= STATE_CLOSE;
				m_ConnectionWatchdog(IN:=FALSE);(*reset connection watchdog*)
				diError := 16#8007;
			END_IF
		0: (* socket was "gracefully closed"  *)
			m_State := STATE_CLOSE;
			diError := 16#8003;
		ELSE (* succesful *)
			m_count:=m_count+m_diReturn;
			IF m_count>=diSendCount THEN
				diError := 16#0000;
				m_State := STATE_RX;
				m_count:=0;
				xStartSend:=FALSE;
			END_IF
			m_ConnectionWatchdog(IN:=FALSE);(*reset connection watchdog*)
		END_CASE


		STATE_CLOSE:	(* Close the server *)

		IF ADR(%MW0)=16#30000000  OR ADR(%MW0)=16#20000000 THEN (*841 or 881*)
			;
		ELSE
			IF m_Socket>=0 THEN
				SysSockShutdown(m_Socket, 0);;(*870*)
			END_IF
		END_IF
		IF m_Socket>=0 THEN
			SysSockClose( m_Socket);
		END_IF
		xClientConnected:= FALSE;
		m_State:= STATE_OPEN; (* Try to open the server again *)
		m_ConnectionWatchdog(IN:=FALSE);(*reset connection watchdog*)

		STATE_ERROR_TRAP: (* Error Read/Write socket  *)
			m_State:= STATE_ERROR_TRAP;

	ELSE  (* Bad FSM code trap  *)
			m_State:= STATE_ERROR_TRAP;
			diError:= 16#8008;
	END_CASE;
ELSE
	IF m_State <> STATE_INIT THEN
		IF ADR(%MW0)=16#30000000  OR ADR(%MW0)=16#20000000 THEN (*841 or 881*)
			;
		ELSE
			IF m_Socket>=0 THEN
				SysSockShutdown(m_Socket, 0);;(*870*)
			END_IF
		END_IF
		IF m_Socket>=0 THEN
			SysSockClose( m_Socket);
		END_IF
		IF ADR(%MW0)=16#30000000  OR ADR(%MW0)=16#20000000 THEN (*841 or 881*)
			;
		ELSE
			IF m_ServerSocket>=0 THEN
				SysSockShutdown(m_ServerSocket, 0);;(*870*)
			END_IF
		END_IF
		IF m_ServerSocket>=0 THEN
			SysSockClose( m_ServerSocket);
		END_IF
		xClientConnected:= FALSE;
		diError:= 0;
		m_State:= STATE_init; (* Try to open the server again *)
		m_ConnectionWatchdog(IN:=FALSE);(*reset connection watchdog*)
	END_IF
END_IF
END_FUNCTION_BLOCK

(* POU TCP_Logger/LogEv, ST *)
FUNCTION LogEv : BOOL
VAR_INPUT
	Level	: en_Logger_ErrLev;
	Object  : en_SYS_Objects;
	Index	: WORD;
	Error	: WORD;
	Message : STRING;
END_VAR
VAR
	s1 : STRING(160);
	i  : INT;
END_VAR
(* Execute error level operations *)
CASE Level OF
	EL_Wrn: 		Sys.Warning:=TRUE;
	EL_Alarm: 		Sys.Alarm  :=TRUE;
	EL_AlarmStop: 	Sys.Alarm  :=TRUE; (* GO TO STOP STATE!! *)
END_CASE

(* Fill lastlog list *)
s1:=CONCAT(Sys.Time_LogString,';Lev=');
s1:=CONCAT(s1,INT_TO_STRING(Level));
s1:=CONCAT(s1,';Obj=');
s1:=CONCAT(s1,INT_TO_STRING(Object));
s1:=CONCAT(s1,';Idx=');
s1:=CONCAT(s1,WORD_TO_STRING(Index));
s1:=CONCAT(s1,';Err=');
s1:=CONCAT(s1,WORD_TO_STRING(Error));
Sys.LastLogs_Dat[Sys.LastLogs_Idx]:=s1;
Sys.LastLogs_Msg[Sys.LastLogs_Idx]:=Message;
Sys.LastLogs_Idx:=Sys.LastLogs_Idx+1;
IF Sys.LastLogs_Idx>5 THEN Sys.LastLogs_Idx:=0; END_IF

(*---------------------------------------------------------------*)
	Logger_Head();
(*---------------------------------------------------------------*)

(* Insert ERR *)
s1:=CONCAT('&ERR=',INT_TO_STRING(Level));
s1:=CONCAT(s1,';');
s1:=CONCAT(s1,INT_TO_STRING(Object));
s1:=CONCAT(s1,';');
s1:=CONCAT(s1,WORD_TO_STRING(Index));
s1:=CONCAT(s1,';');
s1:=CONCAT(s1,WORD_TO_STRING(Error));
s1:=CONCAT(s1,';');
ADDSTRING(ADR(Logger.TData), ADR(s1), Logger.TLen);
s1:=Message;
STR_NOSPACES(ADR(s1));
ADDSTRING(ADR(Logger.TData), ADR(s1), Logger.TLen);

(*---------------------------------------------------------------*)
	Logger_Send();
(*---------------------------------------------------------------*)
END_FUNCTION

(* POU TCP_Logger/Logger_Head, ST *)
FUNCTION Logger_Head : BOOL
VAR
	s1 : STRING(160);
	i  : BYTE;
END_VAR
Logger.TLen:=0;
(* Set GET header *)
ADDSTRING(ADR(Logger.TData), ADR(Logger_GETSTART), Logger.TLen);

(* Insert Header *)
s1:=INSERT('ID=&V=1&D=',DWORD_TO_STRING(Plant_SN),3);
s1:=CONCAT(s1,Sys.Time_LogString);
s1:=CONCAT(s1,'&S=');
IF Sys.Alarm THEN i:=2; ELSIF Sys.Warning THEN i:=1; ELSE i:=0; END_IF
s1:=CONCAT(s1,BYTE_TO_STRING(i));
ADDSTRING(ADR(Logger.TData), ADR(s1), Logger.TLen);
END_FUNCTION

(* POU Utils Functions/ADDSTRING, ST *)
FUNCTION ADDSTRING : BOOL (* Append string to a byte buffer *)
VAR_INPUT
	pTxData: POINTER TO BYTE;
	pString: POINTER TO BYTE;
END_VAR
VAR_IN_OUT
	TxLen: DINT;
END_VAR
VAR
END_VAR
pTxData:=pTxData+TxLen;
WHILE pString^<>0 DO
	pTxData^:=pString^;
	pString:=pString+1;
	pTxData:=pTxData+1;
	TxLen:=TxLen+1;
END_WHILE
END_FUNCTION

(* POU Utils Functions/STR_NOSPACES, ST *)
FUNCTION STR_NOSPACES : BOOL (* Replace spaces and bad chars with allowed ones, used as HTTP-GET validator *)
VAR_INPUT
	pString: POINTER TO BYTE;
END_VAR
VAR
END_VAR
WHILE pString^<>0 DO
	IF pString^=16#20 (* space *) THEN pString^:=16#5F; (*'_'*) END_IF
	pString:=pString+1;
END_WHILE
END_FUNCTION

(* POU TCP_Logger/Logger_Send, ST *)
FUNCTION Logger_Send : BOOL
VAR
	hFile: 	DWORD;
	pos:	DWORD;
END_VAR
(* Finalize string *)
ADDSTRING(ADR(Logger.TData), ADR(Logger_GETEND), Logger.TLen);

(* Read log position *)
pos:=SysFileGetSize(Logger_DataFile);
(* Check log size, bckup and erase if no pending messages *)
IF pos>100000000 (*100M*) THEN
	hFile:=SysFileOpen(Logger_IndexFile,'r');
	IF hFile=0 THEN
		SysFileDelete(Logger_DataFileOld);
		SysFileRename(Logger_DataFile,Logger_DataFileOld);
		pos:=0;
	ELSE
		SysFileClose(hFile);
	END_IF
END_IF
(* Write message on log file *)
hFile:=SysFileOpen(Logger_DataFile,'a');
IF hFile<>0 THEN
	SysFileWrite(hFile, ADR(Logger.TData), Logger.TLen);
	SysFileClose(hFile);
ELSE
	Sys.Warning:=TRUE;
END_IF


(* Check logger status *)
IF Logger.SendReq=FALSE THEN
	(* Set log position for recovery *)
	Logger.SendIdx:=pos;
	(* Copy message data *)
	MEMCPY(ADR(Logger.TData),ADR(Logger.SendData),DINT_TO_WORD(Logger.TLen));
	Logger.SendLen:=Logger.TLen;
	(* Trigger request *)
	Logger.SendReq:=TRUE;
ELSE
	(* Add message position+size in recovery indexes *)
	hFile:=SysFileOpen(Logger_IndexFile,'a');
	SysFileWrite(hFile, ADR(pos), SIZEOF(pos));
	SysFileWrite(hFile, ADR(Logger.TLen), SIZEOF(Logger.TLen));
	SysFileClose(hFile);
END_IF
END_FUNCTION

(* POU Utils Functions/MEMCPY, ST *)
FUNCTION MEMCPY:BOOL
VAR_INPUT
	pSourceAddress:POINTER TO ARRAY[1..2] OF BYTE;
	pDestinationAddress:POINTER TO ARRAY[1..2] OF BYTE;
	BytesToCopy:WORD;
END_VAR
VAR
END_VAR
WHILE (BytesToCopy > 0) DO
	pDestinationAddress^[1]:=pSourceAddress^[1]; (* copy bytes from source to destination *)
	pDestinationAddress:=ADR(pDestinationAddress^[2]); (* increment destination *)
	pSourceAddress:=ADR(pSourceAddress^[2]);(* increment source *)
	BytesToCopy:=BytesToCopy -1; (* decrement number of bytes to copy *)
END_WHILE
END_FUNCTION

(* POU Utils Functions/HEXTORAW, ST *)
FUNCTION HEXTORAW : WORD
VAR_INPUT
	pString		: POINTER TO BYTE;
	StringLen	: WORD;
	pData		: POINTER TO BYTE;
END_VAR
VAR
	xl: WORD;
	xi: WORD;
	xr: BYTE;
END_VAR
xl:=0;
xi:=0;

WHILE xi<StringLen DO

	IF pString^>=97 AND pString^<=102 THEN
		xr := pString^ - 87;
	ELSIF pString^>=65 AND pString^<=70 THEN
		xr := pString^ - 55;
	ELSIF pString^>=48 AND pString^<=57 THEN
		xr := pString^ - 48;
	ELSE
		xr := 16;
	END_IF

	IF xr<16 THEN
		IF (xi AND 1)=0 THEN
			pData^ := xr * 16;
		ELSE
			pData^ := pData^ + xr;
			pData := pData + 1;
			xl := xl + 1;
		END_IF
	END_IF

	xi := xi + 1;
	pString := pString + 1;

END_WHILE

HEXTORAW:=xl;
END_FUNCTION

(* POU Utils/USRLED_Update, ST *)
PROGRAM USRLED_Update
VAR
	OldStatus: en_SYS_Status;

	aFS : ARRAY [0..24] OF FLASHING_SEQUENCE :=
		(Colour:=GREEN,  Frequency:=1,   Relation:=128, Duration:=t#0s,    NextIndex:=0),  (* 0 => RUNNING *)
		(Colour:=ORANGE, Frequency:=1,   Relation:=128, Duration:=t#0s,    NextIndex:=1),  (* 1 => INIT *)
		(Colour:=RED,    Frequency:=4,   Relation:=128, Duration:=t#0s,    NextIndex:=2),  (* 2 => ERROR *)
		(Colour:=RED,    Frequency:=10,  Relation:=128, Duration:=t#0s,    NextIndex:=3),  (* 3 => ALARM *)
		(Colour:=ORANGE, Frequency:=200, Relation:=16,  Duration:=t#100ms, NextIndex:=11), (* 10 *)
		(Colour:=ORANGE, Frequency:=200, Relation:=32,  Duration:=t#100ms, NextIndex:=12),
		(Colour:=ORANGE, Frequency:=200, Relation:=64,  Duration:=t#100ms, NextIndex:=13),
		(Colour:=ORANGE, Frequency:=200, Relation:=128, Duration:=t#100ms, NextIndex:=14),
		(Colour:=ORANGE, Frequency:=200, Relation:=192, Duration:=t#100ms, NextIndex:=15),
		(Colour:=ORANGE, Frequency:=200, Relation:=128, Duration:=t#100ms, NextIndex:=16),
		(Colour:=ORANGE, Frequency:=200, Relation:=64,  Duration:=t#100ms, NextIndex:=17),
		(Colour:=ORANGE, Frequency:=200, Relation:=32,  Duration:=t#100ms, NextIndex:=18),
		(Colour:=ORANGE, Frequency:=200, Relation:=16,  Duration:=t#100ms, NextIndex:=19),
		(Colour:=ORANGE, Frequency:=200, Relation:=8,   Duration:=t#100ms, NextIndex:=10),
		(Colour:=GREEN,  Frequency:=200, Relation:=16,  Duration:=t#100ms, NextIndex:=21), (* 20 *)
		(Colour:=GREEN,  Frequency:=200, Relation:=32,  Duration:=t#100ms, NextIndex:=22),
		(Colour:=GREEN,  Frequency:=200, Relation:=64,  Duration:=t#100ms, NextIndex:=23),
		(Colour:=GREEN,  Frequency:=200, Relation:=128, Duration:=t#100ms, NextIndex:=24),
		(Colour:=GREEN,  Frequency:=200, Relation:=192, Duration:=t#100ms, NextIndex:=25),
		(Colour:=GREEN,  Frequency:=200, Relation:=128, Duration:=t#100ms, NextIndex:=26),
		(Colour:=GREEN,  Frequency:=200, Relation:=64,  Duration:=t#100ms, NextIndex:=27),
		(Colour:=GREEN,  Frequency:=200, Relation:=32,  Duration:=t#100ms, NextIndex:=28),
		(Colour:=GREEN,  Frequency:=200, Relation:=16,  Duration:=t#100ms, NextIndex:=29),
		(Colour:=GREEN,  Frequency:=200, Relation:=8,   Duration:=t#100ms, NextIndex:=20);

	pFS : POINTER TO FLASHING_SEQUENCE;


END_VAR
IF Sys.Status <> OldStatus THEN

	OldStatus:=Sys.Status;

	CASE OldStatus OF

		S_STARTUP:
			pFS:=ADR(aFS);
			SET_FLASHING_SEQUENCE(EN:=TRUE, POINTER_TO_POINTER_TO_ARRAY:=ADR(pFS));
			SET_FLASHING_SEQUENCE_INDEX(EN:=TRUE, IMMEDIATE:=FALSE, INDEX:=1);
			START_FLASHING_SEQUENCE(EN:=TRUE);

		S_RUNNING:
			SET_FLASHING_SEQUENCE_INDEX(EN:=TRUE, IMMEDIATE:=TRUE, INDEX:=0);

	END_CASE

END_IF
END_PROGRAM

(* POU Plant/SCA_Proc, ST *)
PROGRAM SCA_Proc
VAR
	SCA01_5			:FLT_TAP;
	SCA01_6			:FLT_TAP;

	SCA02_1			:FLT_TAP;
	SCA02_2			:FLT_TAP;
	SCA02_3			:FLT_TAP;
	SCA02_4			:FLT_TAP;
	SCA02_5			:FLT_TAP;
	SCA02_6			:FLT_TAP;
	SCA02_7			:FLT_TAP;
	SCA02_8			:FLT_TAP;
	SCA02_9			:FLT_TAP;

	SCA03_1			:FLT_TAP;
	SCA03_2			:FLT_TAP;
	SCA03_3			:FLT_TAP;
	SCA03_4			:FLT_TAP;
	SCA03_5			:FLT_TAP;
	SCA03_6			:FLT_TAP;
	SCA03_7			:FLT_TAP;
	SCA03_8			:FLT_TAP;
	SCA03_9			:FLT_TAP;
	SCA03_10		:FLT_TAP;
	SCA03_11		:FLT_TAP;
	SCA03_12		:FLT_TAP;
	SCA03_13		:FLT_TAP;
	SCA03_14		:FLT_TAP;
	SCA03_15		:FLT_TAP;
	SCA03_16		:FLT_TAP;
	SCA03_17		:FLT_TAP;
	SCA03_18		:FLT_TAP;
	SCA03_19		:FLT_TAP;
	SCA03_20		:FLT_TAP;
	SCA03_21		:FLT_TAP;
	SCA03_22		:FLT_TAP;

	upd : BOOL;
END_VAR
(***** SCA01 *****)
SCA01_1_DO:=SCA01_6.OUT;

SCA01_2_DO:=SCA02_1.OUT;

SCA01_3_DO:=SCA02_3.OUT  OR SCA02_4.OUT  OR SCA02_5.OUT  OR SCA02_6.OUT  OR
			SCA02_8.OUT  OR SCA02_9.OUT;

SCA01_4_DO:=SCA03_1.OUT  OR SCA03_2.OUT  OR SCA03_4.OUT  OR SCA03_6.OUT  OR
			SCA03_8.OUT  OR SCA03_10.OUT OR SCA03_12.OUT OR SCA03_14.OUT OR
			SCA03_16.OUT OR SCA03_18.OUT OR SCA03_20.OUT OR SCA03_22.OUT;

SCA01_5(IN:=NOT SCA01_5_DI);
IF SCA01_5.EVL THEN LogEv(EL_Wrn,EO_SCA,1,1,'5'); upd:=TRUE; END_IF
IF SCA01_5.EVH THEN	LogEv(EL_Log,EO_SCA,1,2,'5'); upd:=TRUE; END_IF

SCA01_6(IN:=NOT SCA01_6_DI);
IF SCA01_6.EVL THEN	LogEv(EL_Wrn,EO_SCA,1,1,'6'); upd:=TRUE; END_IF
IF SCA01_6.EVH THEN	LogEv(EL_Log,EO_SCA,1,2,'6'); upd:=TRUE; END_IF

(***** SCA02 *****)

SCA02_1(IN:=NOT SCA02_1_DI);
IF SCA02_1.EVL THEN	LogEv(EL_Wrn,EO_SCA,2,1,'1'); upd:=TRUE; END_IF
IF SCA02_1.EVH THEN	LogEv(EL_Log,EO_SCA,2,2,'1'); upd:=TRUE; END_IF
SCA02_2(IN:=SCA02_2_DI);
IF SCA02_2.EVL THEN	LogEv(EL_Log,EO_SCA,2,1,'2'); END_IF
IF SCA02_2.EVH THEN	LogEv(EL_Log,EO_SCA,2,2,'2'); END_IF
SCA02_3(IN:=NOT SCA02_3_DI);
IF SCA02_3.EVL THEN	LogEv(EL_Wrn,EO_SCA,2,1,'3'); upd:=TRUE; END_IF
IF SCA02_3.EVH THEN	LogEv(EL_Log,EO_SCA,2,2,'3'); upd:=TRUE; END_IF
SCA02_4(IN:=NOT SCA02_4_DI);
IF SCA02_4.EVL THEN	LogEv(EL_Wrn,EO_SCA,2,1,'4'); upd:=TRUE; END_IF
IF SCA02_4.EVH THEN	LogEv(EL_Log,EO_SCA,2,2,'4'); upd:=TRUE; END_IF
SCA02_5(IN:=NOT SCA02_5_DI);
IF SCA02_5.EVL THEN	LogEv(EL_Wrn,EO_SCA,2,1,'5'); upd:=TRUE; END_IF
IF SCA02_5.EVH THEN	LogEv(EL_Log,EO_SCA,2,2,'5'); upd:=TRUE; END_IF
SCA02_6(IN:=NOT SCA02_6_DI);
IF SCA02_6.EVL THEN	LogEv(EL_Wrn,EO_SCA,2,1,'6'); upd:=TRUE; END_IF
IF SCA02_6.EVH THEN	LogEv(EL_Log,EO_SCA,2,2,'6'); upd:=TRUE; END_IF
SCA02_7(IN:=SCA02_7_DI);
IF SCA02_7.EVL THEN	LogEv(EL_Log,EO_SCA,2,1,'7'); END_IF
IF SCA02_7.EVH THEN	LogEv(EL_Log,EO_SCA,2,2,'7'); END_IF
SCA02_8(IN:=NOT SCA02_8_DI);
IF SCA02_8.EVL THEN	LogEv(EL_Wrn,EO_SCA,2,1,'8'); upd:=TRUE; END_IF
IF SCA02_8.EVH THEN	LogEv(EL_Log,EO_SCA,2,2,'8'); upd:=TRUE; END_IF
SCA02_9(IN:=NOT SCA02_9_DI);
IF SCA02_9.EVL THEN	LogEv(EL_Wrn,EO_SCA,2,1,'9'); upd:=TRUE; END_IF
IF SCA02_9.EVH THEN	LogEv(EL_Log,EO_SCA,2,2,'9'); upd:=TRUE; END_IF

(***** SCA03 *****)

SCA03_1(IN:=NOT SCA03_1_DI);
IF SCA03_1.EVL THEN	LogEv(EL_Wrn,EO_SCA,3,1,'1'); upd:=TRUE; END_IF
IF SCA03_1.EVH THEN	LogEv(EL_Log,EO_SCA,3,2,'1'); upd:=TRUE; END_IF
SCA03_2(IN:=NOT SCA03_2_DI);
IF SCA03_2.EVL THEN	LogEv(EL_Wrn,EO_SCA,3,1,'2'); upd:=TRUE; END_IF
IF SCA03_2.EVH THEN	LogEv(EL_Log,EO_SCA,3,2,'2'); upd:=TRUE; END_IF
SCA03_3(IN:=SCA03_3_DI);
IF SCA03_3.EVL THEN	LogEv(EL_Log,EO_SCA,3,1,'3'); END_IF
IF SCA03_3.EVH THEN	LogEv(EL_Log,EO_SCA,3,2,'3'); END_IF
SCA03_4(IN:=NOT SCA03_4_DI);
IF SCA03_4.EVL THEN	LogEv(EL_Wrn,EO_SCA,3,1,'4'); upd:=TRUE; END_IF
IF SCA03_4.EVH THEN	LogEv(EL_Log,EO_SCA,3,2,'4'); upd:=TRUE; END_IF
SCA03_5(IN:=SCA03_5_DI);
IF SCA03_5.EVL THEN	LogEv(EL_Log,EO_SCA,3,1,'5'); END_IF
IF SCA03_5.EVH THEN	LogEv(EL_Log,EO_SCA,3,2,'5'); END_IF
SCA03_6(IN:=NOT SCA03_6_DI);
IF SCA03_6.EVL THEN	LogEv(EL_Wrn,EO_SCA,3,1,'6'); upd:=TRUE; END_IF
IF SCA03_6.EVH THEN	LogEv(EL_Log,EO_SCA,3,2,'6'); upd:=TRUE; END_IF
SCA03_7(IN:=SCA03_7_DI);
IF SCA03_7.EVL THEN	LogEv(EL_Log,EO_SCA,3,1,'7'); END_IF
IF SCA03_7.EVH THEN	LogEv(EL_Log,EO_SCA,3,2,'7'); END_IF
SCA03_8(IN:=NOT SCA03_8_DI);
IF SCA03_8.EVL THEN	LogEv(EL_Wrn,EO_SCA,3,1,'8'); upd:=TRUE; END_IF
IF SCA03_8.EVH THEN	LogEv(EL_Log,EO_SCA,3,2,'8'); upd:=TRUE; END_IF
SCA03_9(IN:=SCA03_9_DI);
IF SCA03_9.EVL THEN	LogEv(EL_Log,EO_SCA,3,1,'9'); END_IF
IF SCA03_9.EVH THEN	LogEv(EL_Log,EO_SCA,3,2,'9'); END_IF
SCA03_10(IN:=NOT SCA03_10_DI);
IF SCA03_10.EVL THEN	LogEv(EL_Wrn,EO_SCA,3,1,'10'); upd:=TRUE; END_IF
IF SCA03_10.EVH THEN	LogEv(EL_Log,EO_SCA,3,2,'10'); upd:=TRUE; END_IF
SCA03_11(IN:=SCA03_11_DI);
IF SCA03_11.EVL THEN	LogEv(EL_Log,EO_SCA,3,1,'11'); END_IF
IF SCA03_11.EVH THEN	LogEv(EL_Log,EO_SCA,3,2,'11'); END_IF
SCA03_12(IN:=NOT SCA03_12_DI);
IF SCA03_12.EVL THEN	LogEv(EL_Wrn,EO_SCA,3,1,'12'); upd:=TRUE; END_IF
IF SCA03_12.EVH THEN	LogEv(EL_Log,EO_SCA,3,2,'12'); upd:=TRUE; END_IF
SCA03_13(IN:=SCA03_13_DI);
IF SCA03_13.EVL THEN	LogEv(EL_Log,EO_SCA,3,1,'13'); END_IF
IF SCA03_13.EVH THEN	LogEv(EL_Log,EO_SCA,3,2,'13'); END_IF
SCA03_14(IN:=NOT SCA03_14_DI);
IF SCA03_14.EVL THEN	LogEv(EL_Wrn,EO_SCA,3,1,'14'); upd:=TRUE; END_IF
IF SCA03_14.EVH THEN	LogEv(EL_Log,EO_SCA,3,2,'14'); upd:=TRUE; END_IF
SCA03_15(IN:=SCA03_15_DI);
IF SCA03_15.EVL THEN	LogEv(EL_Log,EO_SCA,3,1,'15'); END_IF
IF SCA03_15.EVH THEN	LogEv(EL_Log,EO_SCA,3,2,'15'); END_IF
SCA03_16(IN:=NOT SCA03_16_DI);
IF SCA03_16.EVL THEN	LogEv(EL_Wrn,EO_SCA,3,1,'16'); upd:=TRUE; END_IF
IF SCA03_16.EVH THEN	LogEv(EL_Log,EO_SCA,3,2,'16'); upd:=TRUE; END_IF
SCA03_17(IN:=SCA03_17_DI);
IF SCA03_17.EVL THEN	LogEv(EL_Log,EO_SCA,3,1,'17'); END_IF
IF SCA03_17.EVH THEN	LogEv(EL_Log,EO_SCA,3,2,'17'); END_IF
SCA03_18(IN:=NOT SCA03_18_DI);
IF SCA03_18.EVL THEN	LogEv(EL_Wrn,EO_SCA,3,1,'18'); upd:=TRUE; END_IF
IF SCA03_18.EVH THEN	LogEv(EL_Log,EO_SCA,3,2,'18'); upd:=TRUE; END_IF
SCA03_19(IN:=SCA03_19_DI);
IF SCA03_19.EVL THEN	LogEv(EL_Log,EO_SCA,3,1,'19'); END_IF
IF SCA03_19.EVH THEN	LogEv(EL_Log,EO_SCA,3,2,'19'); END_IF
SCA03_20(IN:=NOT SCA03_20_DI);
IF SCA03_20.EVL THEN	LogEv(EL_Wrn,EO_SCA,3,1,'20'); upd:=TRUE; END_IF
IF SCA03_20.EVH THEN	LogEv(EL_Log,EO_SCA,3,2,'20'); upd:=TRUE; END_IF
SCA03_21(IN:=SCA03_21_DI);
IF SCA03_21.EVL THEN	LogEv(EL_Log,EO_SCA,3,1,'21'); END_IF
IF SCA03_21.EVH THEN	LogEv(EL_Log,EO_SCA,3,2,'21'); END_IF
SCA03_22(IN:=NOT SCA03_22_DI);
IF SCA03_22.EVL THEN	LogEv(EL_Wrn,EO_SCA,3,1,'22'); upd:=TRUE; END_IF
IF SCA03_22.EVH THEN	LogEv(EL_Log,EO_SCA,3,2,'22'); upd:=TRUE; END_IF

IF upd THEN
	upd:=FALSE;
	Logger_Head();
	AddLogData();
	Logger_Send();
END_IF
END_PROGRAM
ACTION AddLogData:
Logger.s1:='&SCA01=';
Logger.s1:=CONCAT(Logger.s1,BYTE_TO_STRING(BOOL_TO_BYTE(SCA01_1_DO))		); Logger.s1:=CONCAT(Logger.s1,';');
Logger.s1:=CONCAT(Logger.s1,BYTE_TO_STRING(BOOL_TO_BYTE(SCA01_2_DO))		); Logger.s1:=CONCAT(Logger.s1,';');
Logger.s1:=CONCAT(Logger.s1,BYTE_TO_STRING(BOOL_TO_BYTE(SCA01_3_DO))		); Logger.s1:=CONCAT(Logger.s1,';');
Logger.s1:=CONCAT(Logger.s1,BYTE_TO_STRING(BOOL_TO_BYTE(SCA01_4_DO))		); Logger.s1:=CONCAT(Logger.s1,';');
Logger.s1:=CONCAT(Logger.s1,BYTE_TO_STRING(BOOL_TO_BYTE(SCA01_5.OUT))		); Logger.s1:=CONCAT(Logger.s1,';');
Logger.s1:=CONCAT(Logger.s1,BYTE_TO_STRING(BOOL_TO_BYTE(SCA01_6.OUT))		);
ADDSTRING(ADR(Logger.TData), ADR(Logger.s1), Logger.TLen);

Logger.s1:='&SCA02=';
Logger.s1:=CONCAT(Logger.s1,BYTE_TO_STRING(BOOL_TO_BYTE(SCA02_1.OUT))		); Logger.s1:=CONCAT(Logger.s1,';');
Logger.s1:=CONCAT(Logger.s1,BYTE_TO_STRING(BOOL_TO_BYTE(SCA02_2.OUT))		); Logger.s1:=CONCAT(Logger.s1,';');
Logger.s1:=CONCAT(Logger.s1,BYTE_TO_STRING(BOOL_TO_BYTE(SCA02_3.OUT))		); Logger.s1:=CONCAT(Logger.s1,';');
Logger.s1:=CONCAT(Logger.s1,BYTE_TO_STRING(BOOL_TO_BYTE(SCA02_4.OUT))		); Logger.s1:=CONCAT(Logger.s1,';');
Logger.s1:=CONCAT(Logger.s1,BYTE_TO_STRING(BOOL_TO_BYTE(SCA02_5.OUT))		); Logger.s1:=CONCAT(Logger.s1,';');
Logger.s1:=CONCAT(Logger.s1,BYTE_TO_STRING(BOOL_TO_BYTE(SCA02_6.OUT))		); Logger.s1:=CONCAT(Logger.s1,';');
Logger.s1:=CONCAT(Logger.s1,BYTE_TO_STRING(BOOL_TO_BYTE(SCA02_7.OUT))		); Logger.s1:=CONCAT(Logger.s1,';');
Logger.s1:=CONCAT(Logger.s1,BYTE_TO_STRING(BOOL_TO_BYTE(SCA02_8.OUT))		); Logger.s1:=CONCAT(Logger.s1,';');
Logger.s1:=CONCAT(Logger.s1,BYTE_TO_STRING(BOOL_TO_BYTE(SCA02_9.OUT))		);
ADDSTRING(ADR(Logger.TData), ADR(Logger.s1), Logger.TLen);

Logger.s1:='&SCA03=';
Logger.s1:=CONCAT(Logger.s1,BYTE_TO_STRING(BOOL_TO_BYTE(SCA03_1.OUT))		); Logger.s1:=CONCAT(Logger.s1,';');
Logger.s1:=CONCAT(Logger.s1,BYTE_TO_STRING(BOOL_TO_BYTE(SCA03_2.OUT))		); Logger.s1:=CONCAT(Logger.s1,';');
Logger.s1:=CONCAT(Logger.s1,BYTE_TO_STRING(BOOL_TO_BYTE(SCA03_3.OUT))		); Logger.s1:=CONCAT(Logger.s1,';');
Logger.s1:=CONCAT(Logger.s1,BYTE_TO_STRING(BOOL_TO_BYTE(SCA03_4.OUT))		); Logger.s1:=CONCAT(Logger.s1,';');
Logger.s1:=CONCAT(Logger.s1,BYTE_TO_STRING(BOOL_TO_BYTE(SCA03_5.OUT))		); Logger.s1:=CONCAT(Logger.s1,';');
Logger.s1:=CONCAT(Logger.s1,BYTE_TO_STRING(BOOL_TO_BYTE(SCA03_6.OUT))		); Logger.s1:=CONCAT(Logger.s1,';');
Logger.s1:=CONCAT(Logger.s1,BYTE_TO_STRING(BOOL_TO_BYTE(SCA03_7.OUT))		); Logger.s1:=CONCAT(Logger.s1,';');
Logger.s1:=CONCAT(Logger.s1,BYTE_TO_STRING(BOOL_TO_BYTE(SCA03_8.OUT))		); Logger.s1:=CONCAT(Logger.s1,';');
Logger.s1:=CONCAT(Logger.s1,BYTE_TO_STRING(BOOL_TO_BYTE(SCA03_9.OUT))		); Logger.s1:=CONCAT(Logger.s1,';');
Logger.s1:=CONCAT(Logger.s1,BYTE_TO_STRING(BOOL_TO_BYTE(SCA03_10.OUT))		); Logger.s1:=CONCAT(Logger.s1,';');
Logger.s1:=CONCAT(Logger.s1,BYTE_TO_STRING(BOOL_TO_BYTE(SCA03_11.OUT))		); Logger.s1:=CONCAT(Logger.s1,';');
Logger.s1:=CONCAT(Logger.s1,BYTE_TO_STRING(BOOL_TO_BYTE(SCA03_12.OUT))		); Logger.s1:=CONCAT(Logger.s1,';');
Logger.s1:=CONCAT(Logger.s1,BYTE_TO_STRING(BOOL_TO_BYTE(SCA03_13.OUT))		); Logger.s1:=CONCAT(Logger.s1,';');
Logger.s1:=CONCAT(Logger.s1,BYTE_TO_STRING(BOOL_TO_BYTE(SCA03_14.OUT))		); Logger.s1:=CONCAT(Logger.s1,';');
Logger.s1:=CONCAT(Logger.s1,BYTE_TO_STRING(BOOL_TO_BYTE(SCA03_15.OUT))		); Logger.s1:=CONCAT(Logger.s1,';');
Logger.s1:=CONCAT(Logger.s1,BYTE_TO_STRING(BOOL_TO_BYTE(SCA03_16.OUT))		); Logger.s1:=CONCAT(Logger.s1,';');
Logger.s1:=CONCAT(Logger.s1,BYTE_TO_STRING(BOOL_TO_BYTE(SCA03_17.OUT))		); Logger.s1:=CONCAT(Logger.s1,';');
Logger.s1:=CONCAT(Logger.s1,BYTE_TO_STRING(BOOL_TO_BYTE(SCA03_18.OUT))		); Logger.s1:=CONCAT(Logger.s1,';');
Logger.s1:=CONCAT(Logger.s1,BYTE_TO_STRING(BOOL_TO_BYTE(SCA03_19.OUT))		); Logger.s1:=CONCAT(Logger.s1,';');
Logger.s1:=CONCAT(Logger.s1,BYTE_TO_STRING(BOOL_TO_BYTE(SCA03_20.OUT))		); Logger.s1:=CONCAT(Logger.s1,';');
Logger.s1:=CONCAT(Logger.s1,BYTE_TO_STRING(BOOL_TO_BYTE(SCA03_21.OUT))		); Logger.s1:=CONCAT(Logger.s1,';');
Logger.s1:=CONCAT(Logger.s1,BYTE_TO_STRING(BOOL_TO_BYTE(SCA03_22.OUT))		);
ADDSTRING(ADR(Logger.TData), ADR(Logger.s1), Logger.TLen);
END_ACTION

(* POU Utils Functions/FLT_TAP, ST *)
FUNCTION_BLOCK FLT_TAP
VAR_INPUT
	IN		: BOOL;
	TAP		: BYTE:=4;
	INITEV	: BOOL:=TRUE;
END_VAR
VAR_OUTPUT
	OUT		: BOOL;
	EVH		: BOOL;
	EVL		: BOOL;
END_VAR
VAR
	init	: BOOL:=FALSE;
	cnt		: BYTE;
END_VAR
EVH:=FALSE;
EVL:=FALSE;

IF NOT init THEN
	init := TRUE;
	IF INITEV THEN
		OUT  := NOT IN;
		cnt  := TAP;
	ELSE
		OUT  := IN;
	END_IF
END_IF

IF OUT<>IN THEN
	cnt:=cnt+1;
	IF cnt>TAP THEN
		OUT:=IN;
		cnt:=0;
		IF OUT THEN EVH:=TRUE; ELSE EVL:=TRUE; END_IF
	END_IF
ELSE
	cnt:=0;
END_IF
END_FUNCTION_BLOCK

(* POU Plant/SYS_Proc, ST *)
PROGRAM SYS_Proc
VAR
(*	fALARM_PB		:FLT_TAP;
	fALARM_TB		:FLT_TAP;
	fALARM_PM		:FLT_TAP; *)

(*	fGZB_ST			:FLT_TAP;  (* GATEWAY ZIGBEE *)*)
(*	fVPN_ST1		:FLT_TAP;  (* VPN CONNECT *)*)
	fVPN_ST2		:FLT_TAP;  (* VPN STATUS *)
(*	fKEY_CT_ST		:FLT_TAP;  (* DOOR1 *)*)
(*	fKEY_SCT_ST		:FLT_TAP;  (* DOOR2 *)*)
	fKEY_QE_ST		:FLT_TAP;  (* DOOR3 *)

END_VAR
(*************** ISPESL *****************)
(*
fALARM_PB(IN:=ALARM_PB);
IF fALARM_PB.EVH THEN
	LogEv(EL_AlarmStop,EO_PBV,1,1,'Over_Pressure_Alarm');
END_IF

fALARM_TB(IN:=ALARM_TB);
IF fALARM_TB.EVH THEN
	LogEv(EL_AlarmStop,EO_TBV,1,1,'Over_Temperature_Alarm');
END_IF

fALARM_PM(IN:=ALARM_PM);
IF fALARM_PM.EVH THEN
	LogEv(EL_AlarmStop,EO_PMV,1,1,'Under_Pressure_Alarm');
END_IF
*)
(****************************************)

(*### VPN Connection Check ###*)(*
fVPN_ST1(IN:=VPN_ST1);
IF fVPN_ST1.EVH THEN
	LogEv(EL_Log,EO_VPN,1,1,'CONNECT_ON');
END_IF
IF fVPN_ST1.EVL THEN
	LogEv(EL_Log,EO_VPN,1,2,'CONNECT_OFF');
END_IF*)

(*### VPN Status Check ###*)
fVPN_ST2(IN:=VPN_ST2);
IF fVPN_ST2.EVH THEN
	LogEv(EL_Log,EO_VPN,1,3,'STATUS_UP');
END_IF
IF fVPN_ST2.EVL THEN
	LogEv(EL_Wrn,EO_VPN,1,4,'STATUS_DOWN');
END_IF

(*### DOOR01 Status Check ###*)(*
fKEY_CT_ST(IN:=KEY_CT_ST);
IF fKEY_CT_ST.EVH THEN
	LogEv(EL_Log,EO_DOOR,1,2,'Centrale_termica_Close');
END_IF
IF fKEY_CT_ST.EVL THEN
	LogEv(EL_Wrn,EO_DOOR,1,1,'Centrale_termica_Open');
END_IF*)

(*### DOOR02 Status Check ###*)(*
fKEY_SCT_ST(IN:=KEY_SCT_ST);
IF fKEY_SCT_ST.EVH THEN
	LogEv(EL_Log,EO_DOOR,2,2,'Sottocentrale_termica_Close');
END_IF
IF fKEY_SCT_ST.EVL THEN
	LogEv(EL_Wrn,EO_DOOR,2,1,'Sottocentrale_termica_Open');
END_IF*)

(*### DOOR03 Status Check ###*)
fKEY_QE_ST(IN:=KEY_QE_ST);
IF fKEY_QE_ST.EVH THEN
	LogEv(EL_Log,EO_DOOR,3,2,'Quadro_Close');
END_IF
IF fKEY_QE_ST.EVL THEN
	LogEv(EL_Wrn,EO_DOOR,3,1,'Quadro_Open');
END_IF
END_PROGRAM

(* POU Utils Functions/AVERAGE_DINT, ST *)
FUNCTION_BLOCK AVERAGE_DINT
VAR_INPUT
	IN: 	DINT;
END_VAR
VAR_OUTPUT
	HI:		DINT;
	AVG:	DINT;
	LOW:	DINT;
	ERR:	BOOL;
END_VAR
VAR
	sum:	REAL;
	cnt:	WORD;
END_VAR
IF cnt>=65000 THEN
	ERR:=TRUE;
	Read();
	sum := sum - DINT_TO_REAL(AVG);
	cnt := cnt - 1;
END_IF

sum := sum + DINT_TO_REAL(IN);
cnt := cnt + 1;

IF IN<LOW THEN LOW:=IN; END_IF
IF IN>HI  THEN HI :=IN; END_IF
END_FUNCTION_BLOCK
ACTION Read:
AVG := REAL_TO_DINT(sum/cnt);
END_ACTION
ACTION Reset:
HI:=IN;
AVG:=IN;
LOW:=IN;
ERR:=FALSE;

sum:=DINT_TO_REAL(IN);
cnt:=1;
END_ACTION

(* POU Utils Functions/AVERAGE_INT, ST *)
FUNCTION_BLOCK AVERAGE_INT
VAR_INPUT
	IN: 	INT;
END_VAR
VAR_OUTPUT
	HI:		INT;
	AVG:	INT;
	LOW:	INT;
	ERR:	BOOL;
END_VAR
VAR
	sum:	DINT;
	cnt:	WORD;
END_VAR
IF cnt>=65000 THEN
	ERR:=TRUE;
	Read();
	sum := sum - AVG;
	cnt := cnt - 1;
END_IF

sum := sum + IN;
cnt := cnt + 1;

IF IN<LOW THEN LOW:=IN; END_IF
IF IN>HI  THEN HI :=IN; END_IF
END_FUNCTION_BLOCK
ACTION Read:
AVG := DINT_TO_INT(sum/cnt);
END_ACTION
ACTION Reset:
HI:=IN;
AVG:=IN;
LOW:=IN;
ERR:=FALSE;

sum:=IN;
cnt:=1;
END_ACTION

(* POU Utils Functions/AVERAGE_T, ST *)
FUNCTION_BLOCK AVERAGE_T
VAR_INPUT
	IN: 	INT;
END_VAR
VAR_OUTPUT
	HI:		INT;
	AVG:	INT;
	LOW:	INT;
	ERR:	BOOL;
END_VAR
VAR
	sum:	DINT;
	cnt:	WORD;
END_VAR
IF cnt>=65000 THEN
	ERR:=TRUE;
	Read();
	sum := sum - AVG;
	cnt := cnt + 1;
END_IF

sum := sum + IN;
cnt := cnt + 1;

IF IN<LOW THEN  LOW:=IN; END_IF
IF IN>HI  THEN HI :=IN; END_IF
END_FUNCTION_BLOCK
ACTION Read:
AVG := DINT_TO_INT(sum/cnt);
END_ACTION
ACTION Reset:
HI:=IN;
AVG:=IN;
LOW:=IN;
ERR:=FALSE;

sum:=IN;
cnt:=1;
END_ACTION

(* POU Utils Functions/COPY_32SWAP16, ST *)
FUNCTION COPY_32SWAP16:BOOL
VAR_INPUT
	pSourceAddress		:POINTER TO ARRAY[1..2] OF WORD;
	pDestinationAddress	:POINTER TO ARRAY[1..2] OF WORD;
END_VAR
VAR
END_VAR
pDestinationAddress^[1]:=pSourceAddress^[2];
pDestinationAddress^[2]:=pSourceAddress^[1];
END_FUNCTION

(* POU Utils/CSV_Log, ST *)
FUNCTION CSV_Log : BOOL
VAR_INPUT
END_VAR
VAR CONSTANT
	LogFileName:STRING:='S:\LOGS_ID3V3.CSV';
END_VAR
VAR
	s1 : STRING(180);
	hFile: 	DWORD;
END_VAR
(* Check file presence *)
hFile:=SysFileOpen(LogFileName,'r');
IF hFile=0 THEN
	(*** File not exist *** Create file and write header *)
	hFile:=SysFileOpen(LogFileName,'w');
	IF hFile<>0 THEN
		(* Write CSV header *)
		s1:='DATE-TIME;T-SA;T-S02;T-S03;T-S04;T-S05;T-S06;T-S07;';
		SysFileWrite(hFile, ADR(s1), LEN(s1));
		s1:='PORT01-Flow;PORT01-Cnt;GAS01-Cnt;GAS02-Cnt;';
		SysFileWrite(hFile, ADR(s1), LEN(s1));
		s1:='CTB250-Power;CTB250-KWH;CTB250-GWH';
		SysFileWrite(hFile, ADR(s1), LEN(s1));
		SysFileWrite(hFile, ADR(Logger_CRLF), LEN(Logger_CRLF));
	END_IF
ELSE
	(*** File exist *** Close file and reopen in append mode *)
	SysFileClose(hFile);
	hFile:=SysFileOpen(LogFileName,'a');
END_IF

(* Log to file *)
IF hFile<>0 THEN
	(* Date stamp *)
	s1:=REPLACE( Sys.Time_LogString , ' ' , 1 , 11 );
	SysFileWrite(hFile, ADR(s1), LEN(s1));
	(* Log data *)
	s1:=CONCAT(';', INT_TO_STRING(TT_S01) );
	s1:=CONCAT(s1 , ';' );
	s1:=CONCAT(s1 , INT_TO_STRING(TPV02.ValoreScalato) );
	s1:=CONCAT(s1 , ';' );
	s1:=CONCAT(s1 , INT_TO_STRING(TPV03.ValoreScalato) );
	s1:=CONCAT(s1 , ';' );
	s1:=CONCAT(s1 , INT_TO_STRING(TPV04.ValoreScalato) );
	s1:=CONCAT(s1 , ';' );
	s1:=CONCAT(s1 , INT_TO_STRING(TPV05.ValoreScalato) );
	s1:=CONCAT(s1 , ';' );
	s1:=CONCAT(s1 , INT_TO_STRING(TPV06.ValoreScalato) );
	s1:=CONCAT(s1 , ';' );
	s1:=CONCAT(s1 , INT_TO_STRING(TPV07.ValoreScalato) );
	SysFileWrite(hFile, ADR(s1), LEN(s1));
	s1:=CONCAT(';', DINT_TO_STRING(PORT01.ValoreScalato/1000) );
	s1:=CONCAT(s1 , ';' );
	s1:=CONCAT(s1 , DINT_TO_STRING(PortataTotalePORT01) );
	s1:=CONCAT(s1 , ';' );
	s1:=CONCAT(s1 , DINT_TO_STRING(PortataTotaleGAS01) );
	s1:=CONCAT(s1 , ';' );
	s1:=CONCAT(s1 , DINT_TO_STRING(PortataTotaleGAS02) );
	SysFileWrite(hFile, ADR(s1), LEN(s1));
	s1:=CONCAT(';', DINT_TO_STRING(REAL_TO_DINT(CTB250.POWER_KW)) );
	s1:=CONCAT(s1 , ';' );
	s1:=CONCAT(s1 , DWORD_TO_STRING(CTB250_ENERGY) );
	SysFileWrite(hFile, ADR(s1), LEN(s1));

	(* Add line CRLF and close *)
	SysFileWrite(hFile, ADR(Logger_CRLF), LEN(Logger_CRLF));
	SysFileClose(hFile);
END_IF
END_FUNCTION

(* POU Utils Functions/FLT_EVENT, ST *)
FUNCTION_BLOCK FLT_EVENT
VAR_INPUT
	IN		: BOOL;
	INITEV	: BOOL:=TRUE;
END_VAR
VAR_OUTPUT
	EVH		: BOOL;
	EVL		: BOOL;
END_VAR
VAR
	init	: BOOL:=FALSE;
	old		: BOOL;
END_VAR
EVH:=FALSE;
EVL:=FALSE;

IF NOT init THEN
	init:=TRUE;
	IF INITEV THEN
		old := NOT IN;
	ELSE
		old := IN;
	END_IF
END_IF

IF old<>IN THEN
	old:=IN;
	IF IN THEN EVH:=TRUE; ELSE EVL:=TRUE; END_IF
END_IF
END_FUNCTION_BLOCK

(* POU Utils Functions/FLT_TIME, ST *)
FUNCTION_BLOCK FLT_TIME
VAR_INPUT
	IN		: BOOL;
	TTAP	: TIME:=T#5s;
	INITEV	: BOOL:=TRUE;
END_VAR
VAR_OUTPUT
	OUT		: BOOL;
	EVH		: BOOL;
	EVL		: BOOL;
END_VAR
VAR
	init	: BOOL:=FALSE;
	timer	: TON;
END_VAR
EVH:=FALSE;
EVL:=FALSE;

IF NOT init THEN
	init := TRUE;
	IF INITEV THEN
		OUT  := NOT IN;
	ELSE
		OUT  := IN;
	END_IF
END_IF

IF OUT<>IN THEN
	timer(IN:=TRUE,PT:=TTAP);
	IF timer.Q THEN
		OUT:=IN;
		timer(IN:=FALSE);
		IF OUT THEN EVH:=TRUE; ELSE EVL:=TRUE; END_IF
	END_IF
ELSE
	timer(IN:=FALSE);
END_IF
END_FUNCTION_BLOCK

(* POU Utils Functions/LINEAR, ST *)
FUNCTION LINEAR : REAL (* Linear interpolation *)
VAR_INPUT
	X_In	: REAL;
	P1_X	: REAL;
	P1_Y	: REAL;
	P2_X	: REAL;
	P2_Y	: REAL;
END_VAR
VAR
END_VAR
LINEAR:=P1_Y+(((P2_Y-P1_Y)*(X_In-P1_X))/(P2_X-P1_X));
END_FUNCTION

(* POU Utils Functions/LINEAR_BAD, ST *)
FUNCTION LINEAR_BAD : INT (* Linear interpolation *)
VAR_INPUT
	PuntoMinX	: INT;
	PuntoMaxX	: INT;
	ValIn		: INT;
	PuntoMinY	: REAL;
	PuntoMaxY	: REAL;
	Decimali	: BYTE;
END_VAR
VAR
	Gain				: REAL;
	PuntoMinX_R			: REAL;
	PuntoMaxX_R			: REAL;
	Linearizzazione_R	: REAL;
END_VAR
PuntoMinX_R:=INT_TO_REAL(PuntoMinX);
PuntoMaxX_R:=INT_TO_REAL(PuntoMaxX);

Gain:=(PuntoMaxX_R-PuntoMinX_R)/(PuntoMaxY-PuntoMinY);	(* Calcolo in guadagno per la linarizzazione *)
Linearizzazione_R:=PuntoMinx+(Gain*(ValIn-PuntoMinY));	(* Ottengo il valore linearizzato *)

LINEAR_BAD:=REAL_TO_INT(Linearizzazione_R*(EXPT(10, Decimali)));  (* Ottengo intero con i decimai voluti *)
END_FUNCTION

(* POU TCP_Logger/LogTrig, ST *)
FUNCTION LogTrig : BOOL
VAR
	s1 : STRING(160);
	i  : BYTE;
END_VAR
(*---------------------------------------------------------------*)
	Logger_Head();
(*---------------------------------------------------------------*)

(* Insert TPVs *)
TPV01.Mean();
s1:=CONCAT('&TPV=',INT_TO_STRING(TPV01.AVG));
TPV01.Mean_Reset();
s1:=CONCAT(s1,';'); s1:=CONCAT(s1,INT_TO_STRING(TPV02.ValoreScalato));
s1:=CONCAT(s1,';'); s1:=CONCAT(s1,INT_TO_STRING(TPV03.ValoreScalato));
s1:=CONCAT(s1,';'); s1:=CONCAT(s1,INT_TO_STRING(TPV04.ValoreScalato));
s1:=CONCAT(s1,';'); s1:=CONCAT(s1,INT_TO_STRING(TPV05.ValoreScalato));
s1:=CONCAT(s1,';'); s1:=CONCAT(s1,INT_TO_STRING(TPV06.ValoreScalato));
s1:=CONCAT(s1,';'); s1:=CONCAT(s1,INT_TO_STRING(TPV07.ValoreScalato));
ADDSTRING(ADR(Logger.TData), ADR(s1), Logger.TLen);

(* Insert contabilizers  *)

s1:=CONCAT('&PORT01=',DINT_TO_STRING(PORT01.ValoreScalato));
s1:=CONCAT(s1,';'); s1:=CONCAT(s1,DINT_TO_STRING(PortataTotalePORT01));
s1:=CONCAT(s1,';'); s1:=CONCAT(s1,BYTE_TO_STRING(PORT01.Status_Log));
ADDSTRING(ADR(Logger.TData), ADR(s1), Logger.TLen);

s1:=CONCAT('&GAS01=',DINT_TO_STRING(PortataTotaleGAS01));
s1:=CONCAT(s1,';'); s1:=CONCAT(s1,BYTE_TO_STRING(GAS01.Status_Log));
ADDSTRING(ADR(Logger.TData), ADR(s1), Logger.TLen);

s1:=CONCAT('&GAS02=',DINT_TO_STRING(PortataTotaleGAS02));
s1:=CONCAT(s1,';'); s1:=CONCAT(s1,BYTE_TO_STRING(GAS02.Status_Log));
ADDSTRING(ADR(Logger.TData), ADR(s1), Logger.TLen);

(*CTBSCAN01.AddLogData( MBUS:=MBUS01 ); ==> TOO BIG! *)
CTB250.AddLogData( ENERGY_WH:=CTB250_ENERGY_WH,	ENERGY:=CTB250_ENERGY );

SCA_Proc.AddLogData();

(*---------------------------------------------------------------*)
	Logger_Send();
(*---------------------------------------------------------------*)
END_FUNCTION

(* POU Utils Functions/MEMCLR, ST *)
FUNCTION MEMCLR:BOOL
VAR_INPUT
	pDestinationAddress:POINTER TO ARRAY[1..2] OF BYTE;
	BytesToClear:WORD;
END_VAR
VAR
END_VAR
WHILE (BytesToClear > 0) DO
	pDestinationAddress^[1]:=0;
	pDestinationAddress:=ADR(pDestinationAddress^[2]); (* increment destination *)
	BytesToClear:=BytesToClear -1; (* decrement number of bytes to copy *)
END_WHILE
END_FUNCTION

(* POU Plant_Objects/obj_GAS, ST *)
FUNCTION_BLOCK obj_GAS
(* === GENERIC PULSE GAS CONTABILIZER ===
   v1.0[23/03/15] - Cleanup and logger action
*)
VAR_INPUT
	(* Settings *)
	ID				: BYTE;			(* Index of instanced object *)
	Peso			: INT:=1;		(* Weight of inpulse [m^3] *)
	TempoTimeOut	: TIME:=T#1m;	(* Activity timeout for warning *)
	(* Physical inputs *)
	GAS_DI			: BOOL;	(* Pulse digital input *)
END_VAR
VAR_IN_OUT
	Contatore       : DINT;
	Totalizzatore	: DINT; (* Totale Conteggio x valore peso *)
END_VAR
VAR_OUTPUT
	(* Status *)
	Status_Log		: BYTE;
	Status_Vis 		: DWORD;
END_VAR
VAR
	Counter			: FLT_TAP := (TAP:=2);
	TimeOut			: TON;
	Warning			: FLT_EVENT;
END_VAR
(* Imposto il time out se non c'è movimento sulla linea per il tempo impostato loggo un Warning *)
TimeOut( IN:=NOT GAS_DI, PT:=TempoTimeOut );

Warning( IN:= TimeOut.Q );

IF Warning.EVH THEN
	(* Condizione di WARNING *)
	Status_Log:=1; Status_Vis:=COLOR_YELLOW;
	LogEv(EL_Wrn,EO_GAS,ID,2,'Nessun_Movimento');
END_IF

IF Warning.EVL THEN
	(* Condizione di Rientro dal WARNING *)
	Status_Log:=0; Status_Vis:=COLOR_GREEN;
	LogEv(EL_Log,EO_GAS,ID,1,'');
END_IF
END_FUNCTION_BLOCK
ACTION Count:
(* Triggero sul fronte di salita l'ingresso digitale *)
Counter(IN:=GAS_DI);

(* Conto i fronti di salita  in modo de creare rapporto*)
IF Counter.EVH THEN
	Contatore:=Contatore+1;
	Totalizzatore:=Contatore*Peso;
END_IF
END_ACTION

(* POU Plant_Objects/obj_MBUS, ST *)
FUNCTION_BLOCK obj_MBUS
(* === M-BUS PROTOCOL INTERFACE ===
   v1.0[16/03/15] - Added interface errors
*)
VAR_INPUT
	(* Settings *)
	ID				: BYTE;
	COM				: BYTE;
	BAUDRATE		: COM_BAUDRATE;
	(* Interface *)
	MBus 			: typMBus;
	MBus_Master 	: FbMBusMaster;
END_VAR
VAR_OUTPUT
	(* Status *)
	Status_Log		: BYTE;
	Status_Vis 		: DWORD;
END_VAR
VAR
	Alarm			: FLT_EVENT;
END_VAR
MBus_Master( bCOMPORT:=COM , enumBAUDRATE:=BAUDRATE , utMBus:=MBus );

(* Check status *)
Alarm(IN:=(MBus.bCOM_ERROR<>0));
IF Alarm.EVH THEN
	LogEv(EL_Alarm,EO_MBUS,ID,1,BYTE_TO_STRING(MBus.bCOM_ERROR));
END_IF
IF Alarm.EVL THEN
	LogEv(EL_Log,EO_MBUS,ID,2,'MBUS_OK');
END_IF

(* Log/visu status *)
   IF Alarm.IN   					THEN Status_Log:=2; Status_Vis:=COLOR_RED;
ELSIF (MBus.bL1_ERROR AND 16#1F)<>0 THEN Status_Log:=1; Status_Vis:=COLOR_YELLOW;
  				 					ELSE Status_Log:=0; Status_Vis:=COLOR_GREEN;
END_IF
END_FUNCTION_BLOCK

(* POU Plant_Objects/obj_MBUS_CTB_SCANNER, ST *)
FUNCTION_BLOCK obj_MBUS_CTB_SCANNER
(* === MBUS HEAT CONTABILIZERS SCANNER & MANAGER ===
   v1.0[16/04/05] - Versioning
   v1.1[29/06/05] - Support for secondary addresses

	> Save/Load of CTB configuration on SD card 'CTBS01.DAT'

*)
VAR_INPUT
	(* Settings *)
	ID				: BYTE;
	EndScanAddress	: BYTE:=250;
	EndlessRescan   : BOOL:=FALSE;
	RefreshPause	: TIME:=t#240s; (* Refresh pause after complete reading cycle *)
	RescanPause		: TIME:=t#30s;  (* Scan pause after successful reading / refresh retry delay *)
	(* Controls *)
	Refresh			: BOOL; (* Enable automatic refresh of detected CTBs *)
	ListLoad		: BOOL:=TRUE; (* Load list from file *)
	ListSave		: BOOL; (* Save list to file *)
	Rescan			: BOOL; (* Perform complete search for list-update *)
END_VAR
VAR_IN_OUT
	MBUS			: obj_MBUS;
END_VAR
VAR_OUTPUT
(*	ConnectedCTBs	: BYTE; (* Number of connected CTBs at last rescan *)*)
	(* Status *)
	Status_Log		: BYTE;
	Status_Vis 		: DWORD;
END_VAR
VAR

	(* Virtual contabilizer for scanner *)
	M1			: FbMBus_Heat := (xSND_NKE:=FALSE);
	M1_Start	: BOOL;
	C1			: FbUnitConverter;
	C1_Err		: BOOL;

	(* Contabilizers data *)
	CTBS		: ARRAY [0..255] OF typ_MBUS_CTBS;

	sta			: BYTE; (* Status: 0:Idle, 1:Wait scan response, 2:Wait refresh response, 3:Wait refresh delay *)
	cnt		 	: BYTE; (* Selection counter *)
	retry		: BYTE; (* Retries counter *)
	pass_cnt 	: BYTE; (* Active counter *)
	dly 	 	: TON;
	s1 		 	: STRING;

	hName	 : STRING;
	hFile	 : DWORD;
	hOK		 : BOOL;
	hCnt	 : BYTE;

END_VAR
CASE sta OF
	0: (*** INIT ***)
		hName:=INSERT('CTBS.DAT',BYTE_TO_STRING(ID),4);
		IF ID<10 THEN hName:=INSERT(hName,'0',4); END_IF
		hName:=CONCAT(FilesPath,hName);
		sta:=1;

	1: (*** Wait actions ***)
		(* Check load request *)
		IF ListLoad THEN
			ListLoad:=FALSE;
			ListLoad_Exe();
			IF hOK THEN
				Refresh:=TRUE;
			END_IF
		END_IF
		(* Check save request *)
		IF ListSave THEN
			ListSave:=FALSE;
			ListSave_Exe();
		END_IF
		(* Check MBUS not busy *)
		IF NOT M1_Start THEN
			IF Rescan THEN
				(* Start scanning - with fast timeout and only one retry *)
				cnt:=0;
				pass_cnt:=0;
				MBUS.MBus_Master.bRetries:=1;
				MBUS.MBus_Master.tTimeout:=T#1000ms;
				M1.dwAdr:=cnt;
				M1_Start:=TRUE;
				CTBS[cnt].Status_Vis:=COLOR_LBLUE;
				sta:=10;
			ELSIF Refresh THEN
				(* Start refresh *)
				cnt:=0;
				retry:=0;
				GoToNextActive();
				IF cnt>EndScanAddress THEN
					Refresh:=FALSE;
				ELSE
					MBUS.MBus_Master.bRetries:=1;
					MBUS.MBus_Master.tTimeout:=T#2000ms;
					M1.dwAdr:=CTBS[cnt].Address;
					M1_Start:=TRUE;
					sta:=20;
				END_IF
			END_IF
		END_IF

	10: (*** PRIMARY SCAN ***)
		IF NOT Rescan THEN
			sta:=1;
		ELSE
			IF NOT M1_Start THEN
				(* Get scan result *)
				UpdateNode();
				(* Next object *)
				cnt:=cnt+1;
				IF cnt>EndScanAddress THEN
					(*ConnectedCTBs:=pass_cnt;*)
					Rescan:=EndlessRescan;
					sta:=1;
				ELSE
					IF CTBS[cnt-1].Present THEN
						(*dly(IN:=FALSE, PT:=RescanPause);*)
						sta:=11;
					ELSE
						M1.dwAdr:=cnt;
						M1_Start:=TRUE;
						CTBS[cnt].Status_Vis:=COLOR_LBLUE;
					END_IF
				END_IF
			END_IF
		END_IF

	11: (*** PRIMARY SCAN DELAY ***)
		dly(IN:=NOT dly.Q, PT:=RescanPause);
		IF dly.Q THEN
			M1.dwAdr:=cnt;
			M1_Start:=TRUE;
			sta:=10;
		END_IF

	20: (*** REFRESH CTBs READING *)
		IF (NOT Refresh) OR Rescan THEN
			sta:=1;
		ELSE
			IF NOT M1_Start THEN
				(* Check result *)
				IF M1.bError<>0 AND retry<2 THEN
					retry:=retry+1;
					sta:=22;
				ELSE
					(* Get scan result *)
					UpdateNode();
					(* Next object *)
					cnt:=cnt+1;
					GoToNextActive();
					retry:=0;
					IF cnt>EndScanAddress THEN
						sta:=21;
						(*dly(IN:=FALSE, PT:=RefreshPause);*)
					ELSE
						M1.dwAdr:=CTBS[cnt].Address;
						M1_Start:=TRUE;
					END_IF
				END_IF
			END_IF
		END_IF

	21: (*** REFRESH CTBs READING - CYCLE PAUSE ***)
		dly(IN:=NOT dly.Q, PT:=RefreshPause);
		IF dly.Q THEN sta:=1; END_IF

	22: (*** REFRESH CTBs READING - RETRY PAUSE ***)
		dly(IN:=NOT dly.Q, PT:=RescanPause);
		IF dly.Q THEN M1_Start:=TRUE; sta:=20; END_IF

ELSE
	sta:=0;
END_CASE

(* Update virtual contabilizer *)
M1( utMBus:=MBUS.MBus , xStart:=M1_Start );
END_FUNCTION_BLOCK
ACTION AddLogData:
;(*
FOR Logger.i1 := 0 TO EndScanAddress  DO
	IF 	CTBSCAN01.NodoMBusPresente[Logger.i1]=TRUE THEN
		Logger.s1:=INSERT('&CTB=',WORD_TO_STRING(Logger.i1),4);
		IF Logger.i1<10 THEN Logger.s1:=INSERT(Logger.s1,'0',4); END_IF
	    Logger.s1:=CONCAT(Logger.s1,'0' (*CTBSCAN01.CTB_utFTemp [Logger.i1].Value*) ); Logger.s1:=CONCAT(Logger.s1,';');
		Logger.s1:=CONCAT(Logger.s1,'0' (*CTBSCAN01.CTB_utRTemp [Logger.i1].Value*) ); Logger.s1:=CONCAT(Logger.s1,';');
		Logger.s1:=CONCAT(Logger.s1,'0' (*CTBSCAN01.CTB_utFlow  [Logger.i1].Value*) ); Logger.s1:=CONCAT(Logger.s1,';');
		Logger.s1:=CONCAT(Logger.s1,'0' (*CTBSCAN01.CTB_utPower [Logger.i1].Value*) ); Logger.s1:=CONCAT(Logger.s1,';');
		Logger.s1:=CONCAT(Logger.s1,'0' (*CTBSCAN01.CTB_utEnergy[Logger.i1].Value*) ); Logger.s1:=CONCAT(Logger.s1,';');
		Logger.s1:=CONCAT(Logger.s1,BYTE_TO_STRING(CTBSCAN01.Status_Log_NodoMBus[Logger.i1]));
		ADDSTRING(ADR(Logger.TData), ADR(Logger.s1), Logger.TLen);
	END_IF
END_FOR
*)
END_ACTION
ACTION GoToNextActive:
WHILE CTBS[cnt].Present <> TRUE AND cnt<=EndScanAddress DO
	cnt:=cnt+1;
END_WHILE
END_ACTION
ACTION ListLoad_Exe:
hOK:=FALSE;
hFile:=SysFileOpen(hName,'r');
IF hFile<>0 THEN
	FOR hCnt := 1 TO EndScanAddress  DO
		SysFileRead(hFile, ADR(CTBS[hCnt].Present), SIZEOF(CTBS[hCnt].Present));
		SysFileRead(hFile, ADR(CTBS[hCnt].Address), SIZEOF(CTBS[hCnt].Address));
		CTBS[hCnt].Status_Vis:=SEL(CTBS[hCnt].Present,COLOR_GREY,COLOR_LBLUE);
	END_FOR
	SysFileClose(hFile);
	hOK:=TRUE;
END_IF
END_ACTION
ACTION ListSave_Exe:
hOK:=FALSE;
hFile:=SysFileOpen(hName,'w');
IF hFile<>0 THEN
	FOR hCnt := 1 TO EndScanAddress  DO
		SysFileWrite(hFile, ADR(CTBS[hCnt].Present), SIZEOF(CTBS[hCnt].Present));
		SysFileWrite(hFile, ADR(CTBS[hCnt].Address), SIZEOF(CTBS[hCnt].Address));
	END_FOR
	SysFileClose(hFile);
	hOK:=TRUE;
END_IF
END_ACTION
ACTION UpdateNode:
(* Save node data *)
CTBS[cnt].NodeError:=M1.bError;
CTBS[cnt].Info:=M1.utMBInfo;
C1(utMBRecord:=M1.utFTemp  , utUnit:=C    , rValue=>CTBS[cnt].Data_FTemp  , xError=>C1_Err );
C1(utMBRecord:=M1.utRTemp  , utUnit:=C    , rValue=>CTBS[cnt].Data_RTemp  , xError=>C1_Err );
C1(utMBRecord:=M1.utFlow   , utUnit:=m3ph , rValue=>CTBS[cnt].Data_Flow   , xError=>C1_Err );
C1(utMBRecord:=M1.utPower  , utUnit:=W    , rValue=>CTBS[cnt].Data_Power  , xError=>C1_Err );
C1(utMBRecord:=M1.utEnergy , utUnit:=kWh  , rValue=>CTBS[cnt].Data_Energy , xError=>C1_Err );

(* Check node status *)
IF CTBS[cnt].NodeError<>0  THEN
	(* se non sono in allarme di comunicazione loggo l'allarme *)
	IF CTBS[cnt].Status_Log<>2 AND sta=20 THEN
		LogEv(EL_Alarm,EO_CTB,cnt,2,CONCAT('Err',BYTE_TO_STRING(CTBS[cnt].NodeError)));
	END_IF
	(*Check rescan mode *)
	IF sta=10 THEN
		(* Disable presence flag & set grey status *)
		CTBS[cnt].Present:=FALSE;
		CTBS[cnt].Address:=0;
		CTBS[cnt].Status_Log:=3;
		CTBS[cnt].Status_Vis:=COLOR_GREY;
	ELSE
		(* Update status *)
		CTBS[cnt].Status_Log:=2;
		CTBS[cnt].Status_Vis:=COLOR_RED;
	END_IF
ELSE
	(* tutto OK Comunizaione andata a buon termine *)
	(* se non sono in allarme di comunicazione loggo l'allarme, ma  se non presente *)
	IF CTBS[cnt].Status_Log<>0 AND sta=20 THEN
		LogEv(EL_Log,EO_CTB,cnt,1,'Nodo_OK');
	END_IF
	(*se sono in fase di rescan memorizzo la presenza del nodo *)
	IF sta=10 THEN
		CTBS[cnt].Present:=TRUE;
		CTBS[cnt].Address:=cnt;
		pass_cnt:=pass_cnt+1;
	END_IF
	(* Update status *)
	CTBS[cnt].Status_Log:=0;
	CTBS[cnt].Status_Vis:=COLOR_GREEN;
END_IF

(* Send data to logger on refresh *)
IF sta=20 THEN
	Logger_Head();
		Logger.s1:=INSERT('&CTB=',WORD_TO_STRING(cnt),4);
		IF cnt<10 THEN Logger.s1:=INSERT(Logger.s1,'0',4); END_IF
	    Logger.s1:=CONCAT(Logger.s1, DINT_TO_STRING(REAL_TO_DINT(CTBS[cnt].Data_FTemp*10  )) ); Logger.s1:=CONCAT(Logger.s1,';');
		Logger.s1:=CONCAT(Logger.s1, DINT_TO_STRING(REAL_TO_DINT(CTBS[cnt].Data_RTemp*10  )) ); Logger.s1:=CONCAT(Logger.s1,';');
		Logger.s1:=CONCAT(Logger.s1, DINT_TO_STRING(REAL_TO_DINT(CTBS[cnt].Data_Flow*1000 )) ); Logger.s1:=CONCAT(Logger.s1,';');
		Logger.s1:=CONCAT(Logger.s1, DINT_TO_STRING(REAL_TO_DINT(CTBS[cnt].Data_Power     )) ); Logger.s1:=CONCAT(Logger.s1,';');
		Logger.s1:=CONCAT(Logger.s1, DINT_TO_STRING(REAL_TO_DINT(CTBS[cnt].Data_Energy/10 )) ); Logger.s1:=CONCAT(Logger.s1,';');
		Logger.s1:=CONCAT(Logger.s1, BYTE_TO_STRING(CTBS[cnt].Status_Log) );
		ADDSTRING(ADR(Logger.TData), ADR(Logger.s1), Logger.TLen);
	Logger_Send();
END_IF

(*VisuDatiMbus[cnt].sdNodoPresente :=SEL(NodoMBusPresente[cnt],'FAIL!','OK'); *)

(* Log found event during scan *)
IF sta=10 AND CTBS[cnt].Present THEN
	s1:='FOUND_';
	s1:=CONCAT(s1, CTBS[cnt].Info.stMED);
	s1:=CONCAT(s1,'_');
	s1:=CONCAT(s1, CTBS[cnt].Info.stID);
	LogEv(EL_Log,EO_CTB,cnt,100,s1);
END_IF
END_ACTION

(* POU Plant_Objects/obj_PORT, ST *)
FUNCTION_BLOCK obj_PORT
(* === FLOW&VOLUME CONTABILIZER ===
   v1.0[16/04/05] - Versioning
*)
VAR_INPUT
	(* Settings *)
	ID			: BYTE;
	Peso		 : INT:=1;		(* Peso dell' impulso , serve per avere una lettura immediata dell'unità ingegneristica *)
	TempoTimeOut : TIME;		(* Minuti di inattività per la segnalazione del WRN *)
	PuntoMinX	: DINT;			(*Parametri per la scalatura *)
	PuntoMaxX	: DINT;
	PuntoMinY	: REAL;
	PuntoMaxY	: REAL;

	TAP			: INT:=2000;   (* Filtro in msec *)
	INITEV		: BOOL:= TRUE; (* Generate init OK event *)
	SogliaHH	: WORD;    (* Soglia per segnalazione Allarme Extra Range in alto - Solitamente sondo in CC *)
	SogliaHL	: WORD;    (* Soglia per segnalazione Allarme Extra Range in Basso - Solitamente sondo Aperta *)
	SogliaWH	: REAL;    (* Soglia per segnalazione Warning  in alto  *)
	SogliaWL	: REAL;    (* Soglia per segnalazione Warning in basso  *)

	(* Physical inputs *)
	DI_INPUT	: BOOL;		(* Ingresso Digitale per il conteggio  *)
	AI_INPUT	: WORD;		(* Ingresso Analogico *)
END_VAR
VAR_IN_OUT
    Contatore		: DINT;
    Totalizzatore	: DINT; (* Totale Conteggio x valore peso *)
END_VAR
VAR_OUTPUT
	ValoreScalato	: DINT;	(* Valore istantaneo scalato ingresso Analgico *)
	ERR				: BOOL;	(* Segnalazione Errore *)
	WRN				: BOOL;	(* Segnalazione Warning *)
	(* Status *)
	Status_Log	: BYTE;
	Status_Vis 	: DWORD;
END_VAR
VAR
	TRig_DI			: R_TRIG;
	TimeOut			: TON;
	TRigR_TimeOut	: R_TRIG;
	TRigL_TimeOut	: F_TRIG;
	SegnaleHH		: BOOL;
	SegnaleHL		: BOOL;
	SegnaleOK		: BOOL;
	SegnaleWH		: BOOL;
	SegnaleWL		: BOOL;
	FiltroWRN		: TON;
	FiltroOK		: TON;
	FiltroERR		: TON;
END_VAR
(*****************************************************************************************)
(**** Gestione ingresso digitale per la contabilizzazzione degli impulsi *****************)
(*****************************************************************************************)

TRig_DI(CLK:=DI_Input );
IF  TRig_DI.Q THEN
	Contatore:=Contatore+1;
	Totalizzatore:=Contatore*Peso;
END_IF

(* Activity monitoring *)
TimeOut(IN:=NOT DI_Input , PT:=TempoTimeOut, Q=> , ET=> );
TRigR_TimeOut(CLK:= TimeOut.Q  );
TRigL_TimeOut(CLK:= TimeOut.Q  );

IF  TRigR_TimeOut.Q THEN
	WRN:=TRUE;
	LogEv(EL_Wrn,EO_PORT,ID,5,'Nessun_Movimento');
END_IF

IF  TRigL_TimeOut.Q THEN
	WRN:=FALSE;
	LogEv(EL_Log,EO_PORT,ID,1,'');
END_IF


(*****************************************************************************************)
(**** Gestione ingresso Analogico per la gestione del valore istantaneo  *****************)
(*****************************************************************************************)

(* Verifico che le variabile letta dall'ingresso Analogico  sia dentro i range
ATTENZIONE I LIMITI SPESSO SONO IN WORD VERIFICA  TABELLA MANUALE WAGO  *)
SegnaleHH:=(AI_INPUT>=SogliaHH);
SegnaleHL:=(AI_INPUT<=SogliaHL);
SegnaleOK:=NOT (SegnaleHH OR SegnaleHL);

(* Linerarizzo il segnale di ingresso e la converto in unita ingegneristiche *)
ValoreScalato:=REAL_TO_DINT(LINEAR( AI_INPUT, PuntoMinY, PuntoMinX, PuntoMaxY, PuntoMaxX ));


IF SegnaleOK  THEN
	(*  Verifica  e segnalazione Warning *)
	SegnaleWH:=(ValoreScalato>SogliaWH);
	SegnaleWL:=(ValoreScalato<SogliaWL);

		FiltroWRN(IN:=(SegnaleWH OR SegnaleWL)  , PT:=INT_TO_TIME(TAP) );    (* Filtro su LOG *)
		IF  FiltroWRN.Q THEN     (* Condizione di WARNING *)
			IF NOT WRN THEN
				WRN:=TRUE;
 				LogEv(EL_Wrn,EO_PORT,ID,SEL(ValoreScalato<=SogliaWL,3,2),DINT_TO_STRING(ValoreScalato));
			END_IF
		END_IF

	IF (INITEV OR WRN OR ERR)  AND NOT FiltroWRN.Q THEN
		FiltroWRN(IN:=FALSE  , PT:=INT_TO_TIME(TAP));    (* Resetto il Filtro su LOG WRN  *)
		FiltroERR(IN:=FALSE  , PT:=INT_TO_TIME(TAP));    (* Resetto il Filtro su LOG ERR *)
		INITEV:=FALSE; ERR:=FALSE; WRN:=FALSE;
		LogEv(EL_Log,EO_PORT,ID,1,'');
	END_IF

	Status_Log:=0;
	Status_Vis:=16#20F020;
ELSE
		FiltroERR(IN:=TRUE , PT:= INT_TO_TIME(TAP) );    (* Filtro su LOG *)
			IF  FiltroERR.Q THEN     (* Condizione di WARNING *)
					IF NOT ERR THEN
						ERR:=TRUE;
						IF SegnaleHH THEN LogEv(EL_Alarm,EO_PORT,ID,6,DINT_TO_STRING(ValoreScalato));END_IF;
						IF SegnaleHL THEN LogEv(EL_Alarm,EO_PORT,ID,4,DINT_TO_STRING(ValoreScalato));END_IF;
					END_IF
			END_IF

	Status_Log:=1;
	Status_Vis:=16#2020F0;
END_IF
END_FUNCTION_BLOCK

(* POU Plant_Objects/obj_SW_CTB, ST *)
FUNCTION_BLOCK obj_SW_CTB
(* === Software Energy contabilizer [TICK=500ms] ===
   v1.0[16/04/05] - Versioning
*)
VAR_INPUT
	(* Settings *)
	ID				: BYTE;
	(* Physical Inputs *)
	T_SEND			: INT;  (* E-1 °C    *)
	T_RET			: INT;  (* E-1 °C    *)
	FLOW			: DINT; (* E-3 m^3/h *)
END_VAR
VAR_IN_OUT
	(* Persistent counter *)
	ENERGY_WH		: REAL;  (* Wh       *)
	ENERGY			: DWORD; (* E-2 MWh  *)
END_VAR
VAR_OUTPUT
	T_SEND_MEAN		: AVERAGE_INT;
	T_RET_MEAN		: AVERAGE_INT;
	FLOW_MEAN		: AVERAGE_DINT;
	POWER_KW		: REAL;
	(* Visu/Log *)
	Status_Log		: BYTE;
	Status_Vis		: DWORD;
END_VAR
VAR
	init			: BOOL;
	overflow		: BOOL;
	P_OLD			: REAL;

	(* HighSpeedLog *)
	hLog  : BOOL   :=FALSE;
	hFile : DWORD  :=0;
	hs1   : STRING;

END_VAR
(* Pv0[kW] = (FLOW/1000) * (8,164 *10 ^ -1 * T_SEND/10 + 9,623*10^2) * 4,186 * (T_SEND - T_RET)/10 / 3600 *)
(*POWER_KW := ( INT_TO_REAL(FLOW) * ( (8.164E-2 * INT_TO_REAL(T_SEND)) + 9.623E2 ) * 4.1868 * (T_SEND-T_RET) ) / 36000 ;*)

(* Pv1[kW] = ( FLOW * (-2.5987E-5 * T_SEND^2 - 1.8693E-2 * T_SEND + 1.0035E3) * 4.1868 * (T_SEND-T_RET) ) / 36E6 *)
POWER_KW := ( DINT_TO_REAL(FLOW) * ( (-2.5987E-5 * EXPT(T_SEND,2)) - (1.8693E-2 * T_SEND) + 1.0035E3 ) * 4.1868 * (T_SEND-T_RET) ) / 36E6 ;

(* Pv2[kW] = ( FLOW * (-2.19E-5 * T_SEND^2 - 2.81E-2 * T_SEND + 1.01E3) * 4.1868 * (T_SEND-T_RET) ) / 36E6 *)
(* ... *)

IF NOT init THEN
	init:=TRUE;
ELSE
	IF (POWER_KW + P_OLD)>0 THEN
		(* E[Wh] = ( (P0+P1)/2 ) * 0,5 / 3600 = (P0+P1)/14400 *)
		ENERGY_WH := ENERGY_WH + (( POWER_KW + P_OLD ) / 14.4);
	END_IF
END_IF

P_OLD:=POWER_KW;

IF ENERGY_WH>10000 THEN
	ENERGY_WH := ENERGY_WH - 10000;
	ENERGY := ENERGY + 1;
END_IF

(* Average of input values *)
T_SEND_MEAN(IN:=T_SEND);
T_RET_MEAN(IN:=T_RET);
FLOW_MEAN(IN:=FLOW);

(* Check status *)
Status_Log:=0; Status_Vis:=16#20F020;

hDbgLog();
END_FUNCTION_BLOCK
ACTION AddLogData:
Logger.s1:=INSERT('&CTB=',BYTE_TO_STRING(ID),4);
IF ID<10 THEN Logger.s1:=INSERT(Logger.s1,'0',4); END_IF
Mean();
Logger.s1:=CONCAT(Logger.s1,INT_TO_STRING(T_SEND_MEAN.AVG)					); Logger.s1:=CONCAT(Logger.s1,';');
Logger.s1:=CONCAT(Logger.s1,INT_TO_STRING(T_RET_MEAN.AVG)					); Logger.s1:=CONCAT(Logger.s1,';');
Logger.s1:=CONCAT(Logger.s1,DINT_TO_STRING(FLOW_MEAN.AVG)					); Logger.s1:=CONCAT(Logger.s1,';');
Mean_Reset();
Logger.s1:=CONCAT(Logger.s1,DINT_TO_STRING(REAL_TO_DINT(POWER_KW*1000))		); Logger.s1:=CONCAT(Logger.s1,';');
Logger.s1:=CONCAT(Logger.s1,DWORD_TO_STRING(ENERGY)							); Logger.s1:=CONCAT(Logger.s1,';');
Logger.s1:=CONCAT(Logger.s1,BYTE_TO_STRING(Status_Log)						);
ADDSTRING(ADR(Logger.TData), ADR(Logger.s1), Logger.TLen);
END_ACTION
ACTION hDbgLog:
IF hLog THEN
	IF hFile=0 THEN
		(* Open file *)
		hFile:=SysFileOpen('S:\HSLOG1.CSV','a');
		(* Start time *)
		hs1:=REPLACE( Sys.Time_LogString , ' ' , 1 , 11 );
		hs1:=CONCAT('>> Start', hs1);
		hs1:=CONCAT(hs1,Logger_CRLF);
		SysFileWrite(hFile, ADR(hs1), LEN(hs1));
		(* Data header *)
		hs1:='T-Send;T-Ret;Port;W;E';
		SysFileWrite(hFile, ADR(hs1), LEN(hs1));
	ELSE
		(* Log data *)
		hs1:=INT_TO_STRING(T_SEND);
		hs1:=CONCAT(hs1 , ';' );
		hs1:=CONCAT(hs1 , INT_TO_STRING(T_RET) );
		hs1:=CONCAT(hs1 , ';' );
		hs1:=CONCAT(hs1 , DINT_TO_STRING(FLOW) );
		hs1:=CONCAT(hs1 , ';' );
		hs1:=CONCAT(hs1 , REAL_TO_STRING(POWER_KW) );
		hs1:=CONCAT(hs1 , ';' );
		hs1:=CONCAT(hs1 , REAL_TO_STRING(ENERGY_WH) );
		hs1:=CONCAT(hs1 , Logger_CRLF );
		SysFileWrite(hFile, ADR(hs1), LEN(hs1));
	END_IF
ELSE
	IF hFile<>0 THEN
		(* Start time *)
		hs1:=REPLACE( Sys.Time_LogString , ' ' , 1 , 11 );
		hs1:=CONCAT('>> Stop', hs1);
		hs1:=CONCAT(hs1,Logger_CRLF);
		SysFileWrite(hFile, ADR(hs1), LEN(hs1));
		(* Close file *)
		SysFileClose(hFile);
		hFile:=0;
	END_IF
END_IF
END_ACTION
ACTION Mean:
T_SEND_MEAN.Read();
T_RET_MEAN.Read();
FLOW_MEAN.Read();
END_ACTION
ACTION Mean_Reset:
T_SEND_MEAN.Reset();
T_RET_MEAN.Reset();
FLOW_MEAN.Reset();
END_ACTION

